LIN {X -286.815,Y -42.863,Z 84.157,A 8.500,B 90.000,C 0.000} C_DIS
LIN {X -286.571,Y -44.464,Z 82.253,A 8.820,B 90.000,C 0.000} C_DIS
LIN {X -286.317,Y -46.071,Z 80.355,A 9.141,B 90.000,C 0.000} C_DIS
LIN {X -286.054,Y -47.677,Z 78.457,A 9.463,B 90.000,C 0.000} C_DIS
LIN {X -285.784,Y -49.269,Z 76.549,A 9.782,B 90.000,C 0.000} C_DIS
LIN {X -285.503,Y -50.872,Z 74.651,A 10.103,B 90.000,C 0.000} C_DIS
LIN {X -285.213,Y -52.473,Z 72.753,A 10.425,B 90.000,C 0.000} C_DIS
LIN {X -284.916,Y -54.061,Z 70.845,A 10.744,B 90.000,C 0.000} C_DIS
LIN {X -284.609,Y -55.658,Z 68.946,A 11.065,B 90.000,C 0.000} C_DIS
LIN {X -284.292,Y -57.253,Z 67.048,A 11.386,B 90.000,C 0.000} C_DIS
LIN {X -284.017,Y -58.605,Z 65.403,A 11.659,B 90.000,C 0.000} C_DIS
LIN {X -283.964,Y -58.859,Z 65.202,A 11.710,B 90.000,C 0.000} C_DIS
LIN {X -283.906,Y -59.138,Z 65.153,A 11.767,B 90.000,C 0.000} C_DIS
LIN {X -283.848,Y -59.418,Z 65.202,A 11.823,B 90.000,C 0.000} C_DIS
LIN {X -283.795,Y -59.671,Z 65.403,A 11.874,B 90.000,C 0.000} C_DIS
LIN {X -283.751,Y -59.880,Z 65.687,A 11.916,B 90.000,C 0.000} C_DIS
LIN {X -283.739,Y -59.937,Z 66.462,A 11.928,B 90.000,C 0.000} C_DIS
LIN {X -283.717,Y -60.038,Z 66.779,A 11.948,B 90.000,C 0.000} C_DIS
LIN {X -283.709,Y -60.077,Z 67.718,A 11.956,B 90.000,C 0.000} C_DIS
LIN {X -283.687,Y -60.180,Z 68.098,A 11.977,B 90.000,C 0.000} C_DIS
LIN {X -283.679,Y -60.218,Z 69.146,A 11.985,B 90.000,C 0.000} C_DIS
LIN {X -283.657,Y -60.321,Z 69.525,A 12.005,B 90.000,C 0.000} C_DIS
LIN {X -283.649,Y -60.360,Z 70.464,A 12.013,B 90.000,C 0.000} C_DIS
LIN {X -283.627,Y -60.462,Z 70.826,A 12.034,B 90.000,C 0.000} C_DIS
LIN {X -283.619,Y -60.501,Z 71.765,A 12.042,B 90.000,C 0.000} C_DIS
LIN {X -283.597,Y -60.603,Z 72.126,A 12.062,B 90.000,C 0.000} C_DIS
LIN {X -283.589,Y -60.643,Z 73.066,A 12.070,B 90.000,C 0.000} C_DIS
LIN {X -283.567,Y -60.745,Z 73.445,A 12.091,B 90.000,C 0.000} C_DIS
LIN {X -283.558,Y -60.784,Z 74.493,A 12.099,B 90.000,C 0.000} C_DIS
LIN {X -283.536,Y -60.886,Z 74.872,A 12.120,B 90.000,C 0.000} C_DIS
LIN {X -283.528,Y -60.925,Z 75.812,A 12.127,B 90.000,C 0.000} C_DIS
LIN {X -283.506,Y -61.028,Z 76.191,A 12.148,B 90.000,C 0.000} C_DIS
LIN {X -283.498,Y -61.066,Z 77.239,A 12.156,B 90.000,C 0.000} C_DIS
LIN {X -283.476,Y -61.169,Z 77.618,A 12.177,B 90.000,C 0.000} C_DIS
LIN {X -283.467,Y -61.208,Z 78.558,A 12.185,B 90.000,C 0.000} C_DIS
LIN {X -283.445,Y -61.310,Z 78.919,A 12.205,B 90.000,C 0.000} C_DIS
LIN {X -283.437,Y -61.349,Z 79.859,A 12.213,B 90.000,C 0.000} C_DIS
LIN {X -283.414,Y -61.451,Z 80.220,A 12.234,B 90.000,C 0.000} C_DIS
LIN {X -283.406,Y -61.490,Z 81.159,A 12.242,B 90.000,C 0.000} C_DIS
LIN {X -283.384,Y -61.592,Z 81.521,A 12.262,B 90.000,C 0.000} C_DIS
LIN {X -283.375,Y -61.632,Z 82.460,A 12.270,B 90.000,C 0.000} C_DIS
LIN {X -283.353,Y -61.734,Z 82.840,A 12.291,B 90.000,C 0.000} C_DIS
LIN {X -283.345,Y -61.773,Z 83.887,A 12.299,B 90.000,C 0.000} C_DIS
LIN {X -283.322,Y -61.875,Z 84.267,A 12.319,B 90.000,C 0.000} C_DIS
LIN {X -283.314,Y -61.914,Z 85.206,A 12.327,B 90.000,C 0.000} C_DIS
LIN {X -283.291,Y -62.016,Z 85.586,A 12.348,B 90.000,C 0.000} C_DIS
LIN {X -283.283,Y -62.055,Z 86.633,A 12.356,B 90.000,C 0.000} C_DIS
LIN {X -283.260,Y -62.157,Z 87.013,A 12.377,B 90.000,C 0.000} C_DIS
LIN {X -283.252,Y -62.196,Z 87.952,A 12.384,B 90.000,C 0.000} C_DIS
LIN {X -283.229,Y -62.298,Z 88.314,A 12.405,B 90.000,C 0.000} C_DIS
LIN {X -283.221,Y -62.338,Z 89.253,A 12.413,B 90.000,C 0.000} C_DIS
LIN {X -283.198,Y -62.440,Z 89.614,A 12.434,B 90.000,C 0.000} C_DIS
LIN {X -283.190,Y -62.479,Z 90.554,A 12.442,B 90.000,C 0.000} C_DIS
LIN {X -283.167,Y -62.581,Z 90.933,A 12.462,B 90.000,C 0.000} C_DIS
LIN {X -283.159,Y -62.620,Z 91.981,A 12.470,B 90.000,C 0.000} C_DIS
LIN {X -283.136,Y -62.722,Z 92.360,A 12.491,B 90.000,C 0.000} C_DIS
LIN {X -283.127,Y -62.761,Z 93.300,A 12.499,B 90.000,C 0.000} C_DIS
LIN {X -283.105,Y -62.863,Z 93.661,A 12.519,B 90.000,C 0.000} C_DIS
LIN {X -283.096,Y -62.902,Z 94.601,A 12.527,B 90.000,C 0.000} C_DIS
LIN {X -283.073,Y -63.004,Z 94.962,A 12.548,B 90.000,C 0.000} C_DIS
LIN {X -283.065,Y -63.043,Z 95.901,A 12.556,B 90.000,C 0.000} C_DIS
LIN {X -283.042,Y -63.145,Z 96.281,A 12.576,B 90.000,C 0.000} C_DIS
LIN {X -283.033,Y -63.184,Z 97.329,A 12.584,B 90.000,C 0.000} C_DIS
LIN {X -283.010,Y -63.286,Z 97.708,A 12.605,B 90.000,C 0.000} C_DIS
LIN {X -283.002,Y -63.325,Z 98.647,A 12.613,B 90.000,C 0.000} C_DIS
LIN {X -282.979,Y -63.427,Z 99.009,A 12.634,B 90.000,C 0.000} C_DIS
LIN {X -282.970,Y -63.466,Z 99.948,A 12.641,B 90.000,C 0.000} C_DIS
LIN {X -282.947,Y -63.568,Z 100.309,A 12.662,B 90.000,C 0.000} C_DIS
LIN {X -282.938,Y -63.607,Z 101.249,A 12.670,B 90.000,C 0.000} C_DIS
LIN {X -282.915,Y -63.709,Z 101.628,A 12.691,B 90.000,C 0.000} C_DIS
LIN {X -282.907,Y -63.748,Z 102.676,A 12.699,B 90.000,C 0.000} C_DIS
LIN {X -282.884,Y -63.850,Z 103.055,A 12.719,B 90.000,C 0.000} C_DIS
LIN {X -282.875,Y -63.889,Z 103.995,A 12.727,B 90.000,C 0.000} C_DIS
LIN {X -282.852,Y -63.991,Z 104.356,A 12.748,B 90.000,C 0.000} C_DIS
LIN {X -282.843,Y -64.030,Z 105.296,A 12.756,B 90.000,C 0.000} C_DIS
LIN {X -282.820,Y -64.132,Z 105.657,A 12.776,B 90.000,C 0.000} C_DIS
LIN {X -282.811,Y -64.171,Z 106.596,A 12.784,B 90.000,C 0.000} C_DIS
LIN {X -282.788,Y -64.273,Z 106.976,A 12.805,B 90.000,C 0.000} C_DIS
LIN {X -282.779,Y -64.312,Z 108.024,A 12.813,B 90.000,C 0.000} C_DIS
LIN {X -282.756,Y -64.414,Z 108.403,A 12.833,B 90.000,C 0.000} C_DIS
LIN {X -282.747,Y -64.453,Z 109.342,A 12.841,B 90.000,C 0.000} C_DIS
LIN {X -282.724,Y -64.555,Z 109.722,A 12.862,B 90.000,C 0.000} C_DIS
LIN {X -282.715,Y -64.594,Z 110.770,A 12.870,B 90.000,C 0.000} C_DIS
LIN {X -282.691,Y -64.696,Z 111.149,A 12.891,B 90.000,C 0.000} C_DIS
LIN {X -282.682,Y -64.735,Z 112.089,A 12.898,B 90.000,C 0.000} C_DIS
LIN {X -282.659,Y -64.837,Z 112.450,A 12.919,B 90.000,C 0.000} C_DIS
LIN {X -282.650,Y -64.876,Z 113.389,A 12.927,B 90.000,C 0.000} C_DIS
LIN {X -282.627,Y -64.978,Z 113.751,A 12.948,B 90.000,C 0.000} C_DIS
LIN {X -282.618,Y -65.017,Z 114.690,A 12.956,B 90.000,C 0.000} C_DIS
LIN {X -282.594,Y -65.118,Z 115.051,A 12.976,B 90.000,C 0.000} C_DIS
LIN {X -282.585,Y -65.157,Z 115.991,A 12.984,B 90.000,C 0.000} C_DIS
LIN {X -282.562,Y -65.259,Z 116.370,A 13.005,B 90.000,C 0.000} C_DIS
LIN {X -282.553,Y -65.298,Z 117.418,A 13.013,B 90.000,C 0.000} C_DIS
LIN {X -282.529,Y -65.400,Z 117.797,A 13.033,B 90.000,C 0.000} C_DIS
LIN {X -282.520,Y -65.439,Z 118.737,A 13.041,B 90.000,C 0.000} C_DIS
LIN {X -282.497,Y -65.541,Z 119.098,A 13.062,B 90.000,C 0.000} C_DIS
LIN {X -282.488,Y -65.580,Z 120.038,A 13.070,B 90.000,C 0.000} C_DIS
LIN {X -282.464,Y -65.682,Z 120.417,A 13.090,B 90.000,C 0.000} C_DIS
LIN {X -282.455,Y -65.720,Z 121.465,A 13.098,B 90.000,C 0.000} C_DIS
LIN {X -282.431,Y -65.822,Z 121.844,A 13.119,B 90.000,C 0.000} C_DIS
LIN {X -282.422,Y -65.861,Z 122.784,A 13.127,B 90.000,C 0.000} C_DIS
LIN {X -282.398,Y -65.963,Z 123.145,A 13.148,B 90.000,C 0.000} C_DIS
LIN {X -282.389,Y -66.002,Z 124.084,A 13.155,B 90.000,C 0.000} C_DIS
LIN {X -282.365,Y -66.104,Z 124.464,A 13.176,B 90.000,C 0.000} C_DIS
LIN {X -282.356,Y -66.143,Z 125.512,A 13.184,B 90.000,C 0.000} C_DIS
LIN {X -282.333,Y -66.245,Z 125.891,A 13.205,B 90.000,C 0.000} C_DIS
LIN {X -282.323,Y -66.284,Z 126.830,A 13.213,B 90.000,C 0.000} C_DIS
LIN {X -282.299,Y -66.385,Z 127.192,A 13.233,B 90.000,C 0.000} C_DIS
LIN {X -282.290,Y -66.424,Z 128.131,A 13.241,B 90.000,C 0.000} C_DIS
LIN {X -282.266,Y -66.526,Z 128.492,A 13.262,B 90.000,C 0.000} C_DIS
LIN {X -282.257,Y -66.565,Z 129.432,A 13.270,B 90.000,C 0.000} C_DIS
LIN {X -282.233,Y -66.667,Z 129.811,A 13.290,B 90.000,C 0.000} C_DIS
LIN {X -282.224,Y -66.705,Z 130.859,A 13.298,B 90.000,C 0.000} C_DIS
LIN {X -282.200,Y -66.807,Z 131.239,A 13.319,B 90.000,C 0.000} C_DIS
LIN {X -282.191,Y -66.846,Z 132.178,A 13.327,B 90.000,C 0.000} C_DIS
LIN {X -282.167,Y -66.948,Z 132.539,A 13.347,B 90.000,C 0.000} C_DIS
LIN {X -282.157,Y -66.987,Z 133.479,A 13.355,B 90.000,C 0.000} C_DIS
LIN {X -282.133,Y -67.089,Z 133.858,A 13.376,B 90.000,C 0.000} C_DIS
LIN {X -282.124,Y -67.127,Z 134.906,A 13.384,B 90.000,C 0.000} C_DIS
LIN {X -282.100,Y -67.229,Z 135.285,A 13.405,B 90.000,C 0.000} C_DIS
LIN {X -282.090,Y -67.268,Z 136.225,A 13.412,B 90.000,C 0.000} C_DIS
LIN {X -282.066,Y -67.370,Z 136.586,A 13.433,B 90.000,C 0.000} C_DIS
LIN {X -282.057,Y -67.409,Z 137.525,A 13.441,B 90.000,C 0.000} C_DIS
LIN {X -282.033,Y -67.510,Z 137.887,A 13.462,B 90.000,C 0.000} C_DIS
LIN {X -282.023,Y -67.549,Z 138.826,A 13.470,B 90.000,C 0.000} C_DIS
LIN {X -281.999,Y -67.651,Z 139.206,A 13.490,B 90.000,C 0.000} C_DIS
LIN {X -281.990,Y -67.690,Z 140.253,A 13.498,B 90.000,C 0.000} C_DIS
LIN {X -281.965,Y -67.791,Z 140.633,A 13.519,B 90.000,C 0.000} C_DIS
LIN {X -281.956,Y -67.830,Z 141.572,A 13.527,B 90.000,C 0.000} C_DIS
LIN {X -281.931,Y -67.932,Z 141.934,A 13.547,B 90.000,C 0.000} C_DIS
LIN {X -281.922,Y -67.971,Z 142.873,A 13.555,B 90.000,C 0.000} C_DIS
LIN {X -281.897,Y -68.073,Z 143.252,A 13.576,B 90.000,C 0.000} C_DIS
LIN {X -281.888,Y -68.111,Z 144.300,A 13.584,B 90.000,C 0.000} C_DIS
LIN {X -281.863,Y -68.213,Z 144.680,A 13.604,B 90.000,C 0.000} C_DIS
LIN {X -281.854,Y -68.252,Z 145.619,A 13.612,B 90.000,C 0.000} C_DIS
LIN {X -281.829,Y -68.353,Z 145.980,A 13.633,B 90.000,C 0.000} C_DIS
LIN {X -281.820,Y -68.392,Z 146.920,A 13.641,B 90.000,C 0.000} C_DIS
LIN {X -281.795,Y -68.494,Z 147.281,A 13.662,B 90.000,C 0.000} C_DIS
LIN {X -281.786,Y -68.533,Z 148.221,A 13.669,B 90.000,C 0.000} C_DIS
LIN {X -281.761,Y -68.635,Z 148.618,A 13.690,B 90.000,C 0.000} C_DIS
LIN {X -281.761,Y -68.635,Z 149.774,A 13.690,B 90.000,C 0.000} C_DIS
LIN {X -281.774,Y -68.583,Z 149.991,A 13.680,B 90.000,C 0.000} C_DIS
LIN {X -281.786,Y -68.533,Z 150.136,A 13.670,B 90.000,C 0.000} C_DIS
LIN {X -281.795,Y -68.493,Z 150.858,A 13.661,B 90.000,C 0.000} C_DIS
LIN {X -281.820,Y -68.393,Z 151.147,A 13.641,B 90.000,C 0.000} C_DIS
LIN {X -281.830,Y -68.353,Z 151.870,A 13.633,B 90.000,C 0.000} C_DIS
LIN {X -281.854,Y -68.252,Z 152.159,A 13.612,B 90.000,C 0.000} C_DIS
LIN {X -281.864,Y -68.212,Z 152.882,A 13.604,B 90.000,C 0.000} C_DIS
LIN {X -281.888,Y -68.112,Z 153.171,A 13.584,B 90.000,C 0.000} C_DIS
LIN {X -281.898,Y -68.072,Z 153.893,A 13.576,B 90.000,C 0.000} C_DIS
LIN {X -281.922,Y -67.971,Z 154.182,A 13.555,B 90.000,C 0.000} C_DIS
LIN {X -281.931,Y -67.931,Z 154.905,A 13.547,B 90.000,C 0.000} C_DIS
LIN {X -281.956,Y -67.831,Z 155.194,A 13.527,B 90.000,C 0.000} C_DIS
LIN {X -281.965,Y -67.791,Z 155.917,A 13.519,B 90.000,C 0.000} C_DIS
LIN {X -281.989,Y -67.690,Z 156.206,A 13.498,B 90.000,C 0.000} C_DIS
LIN {X -281.999,Y -67.650,Z 156.928,A 13.490,B 90.000,C 0.000} C_DIS
LIN {X -282.023,Y -67.550,Z 157.217,A 13.470,B 90.000,C 0.000} C_DIS
LIN {X -282.033,Y -67.510,Z 157.940,A 13.462,B 90.000,C 0.000} C_DIS
LIN {X -282.057,Y -67.409,Z 158.229,A 13.441,B 90.000,C 0.000} C_DIS
LIN {X -282.066,Y -67.369,Z 158.952,A 13.433,B 90.000,C 0.000} C_DIS
LIN {X -282.090,Y -67.269,Z 159.241,A 13.413,B 90.000,C 0.000} C_DIS
LIN {X -282.100,Y -67.229,Z 159.963,A 13.404,B 90.000,C 0.000} C_DIS
LIN {X -282.124,Y -67.128,Z 160.253,A 13.384,B 90.000,C 0.000} C_DIS
LIN {X -282.133,Y -67.088,Z 160.975,A 13.376,B 90.000,C 0.000} C_DIS
LIN {X -282.157,Y -66.987,Z 161.264,A 13.355,B 90.000,C 0.000} C_DIS
LIN {X -282.167,Y -66.947,Z 161.987,A 13.347,B 90.000,C 0.000} C_DIS
LIN {X -282.191,Y -66.847,Z 162.276,A 13.327,B 90.000,C 0.000} C_DIS
LIN {X -282.200,Y -66.807,Z 162.999,A 13.319,B 90.000,C 0.000} C_DIS
LIN {X -282.224,Y -66.706,Z 163.288,A 13.298,B 90.000,C 0.000} C_DIS
LIN {X -282.233,Y -66.666,Z 164.010,A 13.290,B 90.000,C 0.000} C_DIS
LIN {X -282.257,Y -66.566,Z 164.299,A 13.270,B 90.000,C 0.000} C_DIS
LIN {X -282.266,Y -66.525,Z 165.022,A 13.262,B 90.000,C 0.000} C_DIS
LIN {X -282.290,Y -66.425,Z 165.311,A 13.241,B 90.000,C 0.000} C_DIS
LIN {X -282.300,Y -66.385,Z 166.034,A 13.233,B 90.000,C 0.000} C_DIS
LIN {X -282.323,Y -66.285,Z 166.305,A 13.213,B 90.000,C 0.000} C_DIS
LIN {X -282.333,Y -66.244,Z 166.919,A 13.204,B 90.000,C 0.000} C_DIS
LIN {X -282.356,Y -66.143,Z 167.190,A 13.184,B 90.000,C 0.000} C_DIS
LIN {X -282.366,Y -66.103,Z 167.913,A 13.176,B 90.000,C 0.000} C_DIS
LIN {X -282.389,Y -66.002,Z 168.220,A 13.155,B 90.000,C 0.000} C_DIS
LIN {X -282.398,Y -65.963,Z 169.051,A 13.147,B 90.000,C 0.000} C_DIS
LIN {X -282.422,Y -65.862,Z 169.358,A 13.127,B 90.000,C 0.000} C_DIS
LIN {X -282.431,Y -65.822,Z 170.080,A 13.119,B 90.000,C 0.000} C_DIS
LIN {X -282.455,Y -65.721,Z 170.370,A 13.098,B 90.000,C 0.000} C_DIS
LIN {X -282.464,Y -65.681,Z 171.092,A 13.090,B 90.000,C 0.000} C_DIS
LIN {X -282.488,Y -65.580,Z 171.381,A 13.070,B 90.000,C 0.000} C_DIS
LIN {X -282.497,Y -65.540,Z 172.104,A 13.062,B 90.000,C 0.000} C_DIS
LIN {X -282.520,Y -65.440,Z 172.375,A 13.041,B 90.000,C 0.000} C_DIS
LIN {X -282.530,Y -65.399,Z 172.989,A 13.033,B 90.000,C 0.000} C_DIS
LIN {X -282.553,Y -65.299,Z 173.260,A 13.013,B 90.000,C 0.000} C_DIS
LIN {X -282.562,Y -65.259,Z 173.983,A 13.005,B 90.000,C 0.000} C_DIS
LIN {X -282.585,Y -65.158,Z 174.272,A 12.984,B 90.000,C 0.000} C_DIS
LIN {X -282.595,Y -65.118,Z 174.994,A 12.976,B 90.000,C 0.000} C_DIS
LIN {X -282.618,Y -65.017,Z 175.283,A 12.956,B 90.000,C 0.000} C_DIS
LIN {X -282.627,Y -64.977,Z 176.006,A 12.948,B 90.000,C 0.000} C_DIS
LIN {X -282.650,Y -64.876,Z 176.295,A 12.927,B 90.000,C 0.000} C_DIS
LIN {X -282.659,Y -64.836,Z 177.018,A 12.919,B 90.000,C 0.000} C_DIS
LIN {X -282.682,Y -64.735,Z 177.307,A 12.899,B 90.000,C 0.000} C_DIS
LIN {X -282.692,Y -64.695,Z 178.030,A 12.890,B 90.000,C 0.000} C_DIS
LIN {X -282.715,Y -64.595,Z 178.319,A 12.870,B 90.000,C 0.000} C_DIS
LIN {X -282.724,Y -64.554,Z 179.041,A 12.862,B 90.000,C 0.000} C_DIS
LIN {X -282.747,Y -64.454,Z 179.330,A 12.841,B 90.000,C 0.000} C_DIS
LIN {X -282.756,Y -64.413,Z 180.053,A 12.833,B 90.000,C 0.000} C_DIS
LIN {X -282.779,Y -64.313,Z 180.342,A 12.813,B 90.000,C 0.000} C_DIS
LIN {X -282.788,Y -64.272,Z 181.065,A 12.805,B 90.000,C 0.000} C_DIS
LIN {X -282.811,Y -64.172,Z 181.354,A 12.784,B 90.000,C 0.000} C_DIS
LIN {X -282.820,Y -64.132,Z 182.076,A 12.776,B 90.000,C 0.000} C_DIS
LIN {X -282.843,Y -64.031,Z 182.365,A 12.756,B 90.000,C 0.000} C_DIS
LIN {X -282.852,Y -63.991,Z 183.088,A 12.748,B 90.000,C 0.000} C_DIS
LIN {X -282.875,Y -63.890,Z 183.377,A 12.727,B 90.000,C 0.000} C_DIS
LIN {X -282.884,Y -63.850,Z 184.100,A 12.719,B 90.000,C 0.000} C_DIS
LIN {X -282.906,Y -63.749,Z 184.389,A 12.699,B 90.000,C 0.000} C_DIS
LIN {X -282.916,Y -63.709,Z 185.111,A 12.691,B 90.000,C 0.000} C_DIS
LIN {X -282.938,Y -63.608,Z 185.400,A 12.670,B 90.000,C 0.000} C_DIS
LIN {X -282.947,Y -63.568,Z 186.123,A 12.662,B 90.000,C 0.000} C_DIS
LIN {X -282.970,Y -63.467,Z 186.412,A 12.642,B 90.000,C 0.000} C_DIS
LIN {X -282.979,Y -63.427,Z 187.135,A 12.633,B 90.000,C 0.000} C_DIS
LIN {X -283.001,Y -63.326,Z 187.424,A 12.613,B 90.000,C 0.000} C_DIS
LIN {X -283.010,Y -63.286,Z 188.146,A 12.605,B 90.000,C 0.000} C_DIS
LIN {X -283.033,Y -63.185,Z 188.436,A 12.584,B 90.000,C 0.000} C_DIS
LIN {X -283.042,Y -63.145,Z 189.158,A 12.576,B 90.000,C 0.000} C_DIS
LIN {X -283.064,Y -63.044,Z 189.447,A 12.556,B 90.000,C 0.000} C_DIS
LIN {X -283.073,Y -63.003,Z 190.170,A 12.548,B 90.000,C 0.000} C_DIS
LIN {X -283.096,Y -62.903,Z 190.459,A 12.527,B 90.000,C 0.000} C_DIS
LIN {X -283.105,Y -62.862,Z 191.182,A 12.519,B 90.000,C 0.000} C_DIS
LIN {X -283.127,Y -62.762,Z 191.471,A 12.499,B 90.000,C 0.000} C_DIS
LIN {X -283.136,Y -62.721,Z 192.193,A 12.491,B 90.000,C 0.000} C_DIS
LIN {X -283.158,Y -62.620,Z 192.482,A 12.470,B 90.000,C 0.000} C_DIS
LIN {X -283.167,Y -62.580,Z 193.205,A 12.462,B 90.000,C 0.000} C_DIS
LIN {X -283.190,Y -62.479,Z 193.494,A 12.442,B 90.000,C 0.000} C_DIS
LIN {X -283.198,Y -62.439,Z 194.217,A 12.434,B 90.000,C 0.000} C_DIS
LIN {X -283.221,Y -62.338,Z 194.506,A 12.413,B 90.000,C 0.000} C_DIS
LIN {X -283.230,Y -62.298,Z 195.228,A 12.405,B 90.000,C 0.000} C_DIS
LIN {X -283.252,Y -62.197,Z 195.517,A 12.385,B 90.000,C 0.000} C_DIS
LIN {X -283.261,Y -62.157,Z 196.240,A 12.376,B 90.000,C 0.000} C_DIS
LIN {X -283.283,Y -62.056,Z 196.529,A 12.356,B 90.000,C 0.000} C_DIS
LIN {X -283.291,Y -62.016,Z 197.252,A 12.348,B 90.000,C 0.000} C_DIS
LIN {X -283.314,Y -61.915,Z 197.541,A 12.327,B 90.000,C 0.000} C_DIS
LIN {X -283.322,Y -61.874,Z 198.263,A 12.319,B 90.000,C 0.000} C_DIS
LIN {X -283.344,Y -61.773,Z 198.553,A 12.299,B 90.000,C 0.000} C_DIS
LIN {X -283.353,Y -61.733,Z 199.275,A 12.291,B 90.000,C 0.000} C_DIS
LIN {X -283.375,Y -61.632,Z 199.564,A 12.270,B 90.000,C 0.000} C_DIS
LIN {X -283.384,Y -61.592,Z 200.287,A 12.262,B 90.000,C 0.000} C_DIS
LIN {X -283.406,Y -61.491,Z 200.576,A 12.242,B 90.000,C 0.000} C_DIS
LIN {X -283.415,Y -61.451,Z 201.299,A 12.234,B 90.000,C 0.000} C_DIS
LIN {X -283.436,Y -61.350,Z 201.588,A 12.213,B 90.000,C 0.000} C_DIS
LIN {X -283.445,Y -61.309,Z 202.310,A 12.205,B 90.000,C 0.000} C_DIS
LIN {X -283.467,Y -61.209,Z 202.599,A 12.185,B 90.000,C 0.000} C_DIS
LIN {X -283.476,Y -61.168,Z 203.322,A 12.177,B 90.000,C 0.000} C_DIS
LIN {X -283.497,Y -61.067,Z 203.611,A 12.156,B 90.000,C 0.000} C_DIS
LIN {X -283.506,Y -61.027,Z 204.334,A 12.148,B 90.000,C 0.000} C_DIS
LIN {X -283.528,Y -60.926,Z 204.623,A 12.128,B 90.000,C 0.000} C_DIS
LIN {X -283.537,Y -60.886,Z 205.345,A 12.119,B 90.000,C 0.000} C_DIS
LIN {X -283.558,Y -60.785,Z 205.634,A 12.099,B 90.000,C 0.000} C_DIS
LIN {X -283.567,Y -60.744,Z 206.357,A 12.091,B 90.000,C 0.000} C_DIS
LIN {X -283.588,Y -60.643,Z 206.646,A 12.070,B 90.000,C 0.000} C_DIS
LIN {X -283.597,Y -60.603,Z 207.369,A 12.062,B 90.000,C 0.000} C_DIS
LIN {X -283.619,Y -60.502,Z 207.658,A 12.042,B 90.000,C 0.000} C_DIS
LIN {X -283.627,Y -60.462,Z 208.380,A 12.034,B 90.000,C 0.000} C_DIS
LIN {X -283.649,Y -60.361,Z 208.670,A 12.013,B 90.000,C 0.000} C_DIS
LIN {X -283.657,Y -60.320,Z 209.392,A 12.005,B 90.000,C 0.000} C_DIS
LIN {X -283.679,Y -60.219,Z 209.681,A 11.985,B 90.000,C 0.000} C_DIS
LIN {X -283.687,Y -60.179,Z 210.404,A 11.977,B 90.000,C 0.000} C_DIS
LIN {X -283.709,Y -60.078,Z 210.693,A 11.956,B 90.000,C 0.000} C_DIS
LIN {X -283.717,Y -60.037,Z 211.416,A 11.948,B 90.000,C 0.000} C_DIS
LIN {X -283.739,Y -59.937,Z 211.687,A 11.928,B 90.000,C 0.000} C_DIS
LIN {X -283.747,Y -59.896,Z 212.301,A 11.919,B 90.000,C 0.000} C_DIS
LIN {X -283.769,Y -59.795,Z 212.590,A 11.899,B 90.000,C 0.000} C_DIS
LIN {X -283.777,Y -59.755,Z 213.421,A 11.891,B 90.000,C 0.000} C_DIS
LIN {X -283.798,Y -59.654,Z 213.710,A 11.871,B 90.000,C 0.000} C_DIS
LIN {X -283.807,Y -59.613,Z 214.324,A 11.862,B 90.000,C 0.000} C_DIS
LIN {X -283.828,Y -59.512,Z 214.613,A 11.842,B 90.000,C 0.000} C_DIS
LIN {X -283.836,Y -59.472,Z 215.444,A 11.834,B 90.000,C 0.000} C_DIS
LIN {X -283.858,Y -59.371,Z 215.751,A 11.813,B 90.000,C 0.000} C_DIS
LIN {X -283.866,Y -59.330,Z 216.474,A 11.805,B 90.000,C 0.000} C_DIS
LIN {X -283.887,Y -59.229,Z 216.763,A 11.785,B 90.000,C 0.000} C_DIS
LIN {X -283.896,Y -59.189,Z 217.486,A 11.777,B 90.000,C 0.000} C_DIS
LIN {X -283.917,Y -59.088,Z 217.775,A 11.756,B 90.000,C 0.000} C_DIS
LIN {X -283.925,Y -59.047,Z 218.497,A 11.748,B 90.000,C 0.000} C_DIS
LIN {X -283.946,Y -58.946,Z 218.786,A 11.728,B 90.000,C 0.000} C_DIS
LIN {X -283.954,Y -58.906,Z 219.509,A 11.720,B 90.000,C 0.000} C_DIS
LIN {X -283.975,Y -58.805,Z 219.780,A 11.699,B 90.000,C 0.000} C_DIS
LIN {X -283.984,Y -58.764,Z 220.394,A 11.691,B 90.000,C 0.000} C_DIS
LIN {X -284.005,Y -58.663,Z 220.665,A 11.671,B 90.000,C 0.000} C_DIS
LIN {X -284.013,Y -58.623,Z 221.388,A 11.663,B 90.000,C 0.000} C_DIS
LIN {X -284.034,Y -58.522,Z 221.677,A 11.642,B 90.000,C 0.000} C_DIS
LIN {X -284.042,Y -58.481,Z 222.400,A 11.634,B 90.000,C 0.000} C_DIS
LIN {X -284.063,Y -58.380,Z 222.689,A 11.614,B 90.000,C 0.000} C_DIS
LIN {X -284.071,Y -58.340,Z 223.411,A 11.605,B 90.000,C 0.000} C_DIS
LIN {X -284.092,Y -58.239,Z 223.700,A 11.585,B 90.000,C 0.000} C_DIS
LIN {X -284.100,Y -58.198,Z 224.423,A 11.577,B 90.000,C 0.000} C_DIS
LIN {X -284.121,Y -58.097,Z 224.712,A 11.557,B 90.000,C 0.000} C_DIS
LIN {X -284.129,Y -58.056,Z 225.435,A 11.548,B 90.000,C 0.000} C_DIS
LIN {X -284.150,Y -57.955,Z 225.724,A 11.528,B 90.000,C 0.000} C_DIS
LIN {X -284.158,Y -57.915,Z 226.446,A 11.520,B 90.000,C 0.000} C_DIS
LIN {X -284.179,Y -57.814,Z 226.736,A 11.499,B 90.000,C 0.000} C_DIS
LIN {X -284.187,Y -57.773,Z 227.458,A 11.491,B 90.000,C 0.000} C_DIS
LIN {X -284.208,Y -57.672,Z 227.747,A 11.471,B 90.000,C 0.000} C_DIS
LIN {X -284.216,Y -57.632,Z 228.470,A 11.463,B 90.000,C 0.000} C_DIS
LIN {X -284.236,Y -57.530,Z 228.759,A 11.442,B 90.000,C 0.000} C_DIS
LIN {X -284.244,Y -57.490,Z 229.482,A 11.434,B 90.000,C 0.000} C_DIS
LIN {X -284.265,Y -57.389,Z 229.771,A 11.414,B 90.000,C 0.000} C_DIS
LIN {X -284.273,Y -57.348,Z 230.493,A 11.406,B 90.000,C 0.000} C_DIS
LIN {X -284.293,Y -57.247,Z 230.782,A 11.385,B 90.000,C 0.000} C_DIS
LIN {X -284.302,Y -57.207,Z 231.505,A 11.377,B 90.000,C 0.000} C_DIS
LIN {X -284.322,Y -57.105,Z 231.794,A 11.357,B 90.000,C 0.000} C_DIS
LIN {X -284.330,Y -57.065,Z 232.517,A 11.348,B 90.000,C 0.000} C_DIS
LIN {X -284.350,Y -56.964,Z 232.806,A 11.328,B 90.000,C 0.000} C_DIS
LIN {X -284.358,Y -56.923,Z 233.528,A 11.320,B 90.000,C 0.000} C_DIS
LIN {X -284.379,Y -56.822,Z 233.817,A 11.300,B 90.000,C 0.000} C_DIS
LIN {X -284.387,Y -56.781,Z 234.540,A 11.291,B 90.000,C 0.000} C_DIS
LIN {X -284.407,Y -56.680,Z 234.829,A 11.271,B 90.000,C 0.000} C_DIS
LIN {X -284.415,Y -56.640,Z 235.552,A 11.263,B 90.000,C 0.000} C_DIS
LIN {X -284.425,Y -56.589,Z 235.696,A 11.253,B 90.000,C 0.000} C_DIS
LIN {X -284.435,Y -56.539,Z 235.772,A 11.243,B 90.000,C 0.000} C_DIS
LIN {X -284.448,Y -56.472,Z 236.202,A 11.229,B 90.000,C 0.000} C_DIS
LIN {X -284.474,Y -56.342,Z 236.395,A 11.203,B 90.000,C 0.000} C_DIS
LIN {X -284.514,Y -56.141,Z 236.519,A 11.162,B 90.000,C 0.000} C_DIS
LIN {X -284.565,Y -55.882,Z 236.563,A 11.110,B 90.000,C 0.000} C_DIS
LIN {X -284.623,Y -55.588,Z 236.506,A 11.051,B 90.000,C 0.000} C_DIS
LIN {X -284.683,Y -55.275,Z 236.240,A 10.988,B 90.000,C 0.000} C_DIS
LIN {X -284.727,Y -55.051,Z 235.979,A 10.943,B 90.000,C 0.000} C_DIS
LIN {X -284.745,Y -54.958,Z 235.807,A 10.924,B 90.000,C 0.000} C_DIS
LIN {X -284.749,Y -54.937,Z 235.729,A 10.920,B 90.000,C 0.000} C_DIS
LIN {X -284.768,Y -54.837,Z 235.659,A 10.900,B 90.000,C 0.000} C_DIS
LIN {X -284.772,Y -54.816,Z 235.568,A 10.896,B 90.000,C 0.000} C_DIS
LIN {X -284.780,Y -54.774,Z 235.446,A 10.887,B 90.000,C 0.000} C_DIS
LIN {X -284.819,Y -54.574,Z 235.228,A 10.847,B 90.000,C 0.000} C_DIS
LIN {X -284.835,Y -54.491,Z 235.008,A 10.830,B 90.000,C 0.000} C_DIS
LIN {X -284.873,Y -54.290,Z 234.795,A 10.790,B 90.000,C 0.000} C_DIS
LIN {X -284.889,Y -54.207,Z 234.574,A 10.773,B 90.000,C 0.000} C_DIS
LIN {X -284.927,Y -54.006,Z 234.361,A 10.733,B 90.000,C 0.000} C_DIS
LIN {X -284.943,Y -53.923,Z 234.141,A 10.716,B 90.000,C 0.000} C_DIS
LIN {X -284.981,Y -53.722,Z 233.928,A 10.676,B 90.000,C 0.000} C_DIS
LIN {X -284.996,Y -53.639,Z 233.707,A 10.659,B 90.000,C 0.000} C_DIS
LIN {X -285.034,Y -53.438,Z 233.489,A 10.619,B 90.000,C 0.000} C_DIS
LIN {X -285.042,Y -53.396,Z 233.368,A 10.610,B 90.000,C 0.000} C_DIS
LIN {X -285.046,Y -53.375,Z 233.277,A 10.606,B 90.000,C 0.000} C_DIS
LIN {X -285.065,Y -53.275,Z 233.202,A 10.586,B 90.000,C 0.000} C_DIS
LIN {X -285.068,Y -53.254,Z 233.111,A 10.582,B 90.000,C 0.000} C_DIS
LIN {X -285.076,Y -53.212,Z 232.989,A 10.573,B 90.000,C 0.000} C_DIS
LIN {X -285.114,Y -53.012,Z 232.771,A 10.533,B 90.000,C 0.000} C_DIS
LIN {X -285.129,Y -52.928,Z 232.551,A 10.516,B 90.000,C 0.000} C_DIS
LIN {X -285.166,Y -52.728,Z 232.338,A 10.476,B 90.000,C 0.000} C_DIS
LIN {X -285.182,Y -52.644,Z 232.117,A 10.459,B 90.000,C 0.000} C_DIS
LIN {X -285.219,Y -52.443,Z 231.904,A 10.419,B 90.000,C 0.000} C_DIS
LIN {X -285.234,Y -52.360,Z 231.684,A 10.402,B 90.000,C 0.000} C_DIS
LIN {X -285.271,Y -52.159,Z 231.466,A 10.362,B 90.000,C 0.000} C_DIS
LIN {X -285.278,Y -52.117,Z 231.345,A 10.353,B 90.000,C 0.000} C_DIS
LIN {X -285.282,Y -52.096,Z 231.254,A 10.349,B 90.000,C 0.000} C_DIS
LIN {X -285.301,Y -51.996,Z 231.178,A 10.329,B 90.000,C 0.000} C_DIS
LIN {X -285.304,Y -51.975,Z 231.087,A 10.325,B 90.000,C 0.000} C_DIS
LIN {X -285.312,Y -51.933,Z 230.966,A 10.316,B 90.000,C 0.000} C_DIS
LIN {X -285.348,Y -51.732,Z 230.748,A 10.276,B 90.000,C 0.000} C_DIS
LIN {X -285.364,Y -51.649,Z 230.528,A 10.259,B 90.000,C 0.000} C_DIS
LIN {X -285.400,Y -51.448,Z 230.314,A 10.219,B 90.000,C 0.000} C_DIS
LIN {X -285.415,Y -51.364,Z 230.094,A 10.202,B 90.000,C 0.000} C_DIS
LIN {X -285.451,Y -51.163,Z 229.881,A 10.162,B 90.000,C 0.000} C_DIS
LIN {X -285.466,Y -51.080,Z 229.661,A 10.145,B 90.000,C 0.000} C_DIS
LIN {X -285.502,Y -50.879,Z 229.447,A 10.105,B 90.000,C 0.000} C_DIS
LIN {X -285.517,Y -50.795,Z 229.227,A 10.088,B 90.000,C 0.000} C_DIS
LIN {X -285.552,Y -50.594,Z 229.009,A 10.047,B 90.000,C 0.000} C_DIS
LIN {X -285.560,Y -50.552,Z 228.888,A 10.039,B 90.000,C 0.000} C_DIS
LIN {X -285.564,Y -50.532,Z 228.797,A 10.035,B 90.000,C 0.000} C_DIS
LIN {X -285.581,Y -50.431,Z 228.721,A 10.015,B 90.000,C 0.000} C_DIS
LIN {X -285.585,Y -50.410,Z 228.630,A 10.010,B 90.000,C 0.000} C_DIS
LIN {X -285.592,Y -50.368,Z 228.509,A 10.002,B 90.000,C 0.000} C_DIS
LIN {X -285.628,Y -50.167,Z 228.291,A 9.962,B 90.000,C 0.000} C_DIS
LIN {X -285.642,Y -50.084,Z 228.071,A 9.945,B 90.000,C 0.000} C_DIS
LIN {X -285.678,Y -49.883,Z 227.857,A 9.905,B 90.000,C 0.000} C_DIS
LIN {X -285.692,Y -49.799,Z 227.637,A 9.888,B 90.000,C 0.000} C_DIS
LIN {X -285.727,Y -49.598,Z 227.424,A 9.848,B 90.000,C 0.000} C_DIS
LIN {X -285.742,Y -49.514,Z 227.204,A 9.831,B 90.000,C 0.000} C_DIS
LIN {X -285.777,Y -49.313,Z 226.986,A 9.790,B 90.000,C 0.000} C_DIS
LIN {X -285.784,Y -49.271,Z 226.864,A 9.782,B 90.000,C 0.000} C_DIS
LIN {X -285.787,Y -49.250,Z 226.773,A 9.778,B 90.000,C 0.000} C_DIS
LIN {X -285.805,Y -49.150,Z 226.698,A 9.758,B 90.000,C 0.000} C_DIS
LIN {X -285.808,Y -49.129,Z 226.607,A 9.753,B 90.000,C 0.000} C_DIS
LIN {X -285.815,Y -49.087,Z 226.486,A 9.745,B 90.000,C 0.000} C_DIS
LIN {X -285.850,Y -48.886,Z 226.268,A 9.705,B 90.000,C 0.000} C_DIS
LIN {X -285.864,Y -48.802,Z 226.047,A 9.688,B 90.000,C 0.000} C_DIS
LIN {X -285.899,Y -48.601,Z 225.829,A 9.648,B 90.000,C 0.000} C_DIS
LIN {X -285.906,Y -48.559,Z 225.708,A 9.639,B 90.000,C 0.000} C_DIS
LIN {X -285.914,Y -48.511,Z 225.608,A 9.630,B 90.000,C 0.000} C_DIS
LIN {X -285.942,Y -48.345,Z 225.579,A 9.596,B 90.000,C 0.000} C_DIS
LIN {X -285.967,Y -48.194,Z 225.601,A 9.566,B 90.000,C 0.000} C_DIS
LIN {X -285.978,Y -48.131,Z 225.652,A 9.554,B 90.000,C 0.000} C_DIS
LIN {X -285.992,Y -48.048,Z 225.703,A 9.537,B 90.000,C 0.000} C_DIS
LIN {X -286.026,Y -47.846,Z 225.724,A 9.496,B 90.000,C 0.000} C_DIS
LIN {X -286.059,Y -47.645,Z 225.703,A 9.456,B 90.000,C 0.000} C_DIS
LIN {X -286.073,Y -47.561,Z 225.652,A 9.439,B 90.000,C 0.000} C_DIS
LIN {X -286.079,Y -47.528,Z 225.601,A 9.433,B 90.000,C 0.000} C_DIS
LIN {X -286.110,Y -47.339,Z 225.550,A 9.395,B 90.000,C 0.000} C_DIS
LIN {X -286.127,Y -47.237,Z 225.474,A 9.375,B 90.000,C 0.000} C_DIS
LIN {X -286.139,Y -47.162,Z 225.371,A 9.360,B 90.000,C 0.000} C_DIS
LIN {X -286.148,Y -47.112,Z 225.179,A 9.350,B 90.000,C 0.000} C_DIS
LIN {X -286.156,Y -47.062,Z 225.146,A 9.339,B 90.000,C 0.000} C_DIS
LIN {X -286.164,Y -47.012,Z 225.040,A 9.329,B 90.000,C 0.000} C_DIS
LIN {X -286.171,Y -46.970,Z 224.529,A 9.321,B 90.000,C 0.000} C_DIS
LIN {X -286.179,Y -46.919,Z 224.423,A 9.311,B 90.000,C 0.000} C_DIS
LIN {X -286.188,Y -46.869,Z 224.279,A 9.301,B 90.000,C 0.000} C_DIS
LIN {X -286.194,Y -46.828,Z 223.556,A 9.293,B 90.000,C 0.000} C_DIS
LIN {X -286.203,Y -46.777,Z 223.411,A 9.282,B 90.000,C 0.000} C_DIS
LIN {X -286.211,Y -46.726,Z 223.310,A 9.272,B 90.000,C 0.000} C_DIS
LIN {X -286.219,Y -46.675,Z 222.773,A 9.262,B 90.000,C 0.000} C_DIS
LIN {X -286.237,Y -46.563,Z 222.617,A 9.239,B 90.000,C 0.000} C_DIS
LIN {X -286.254,Y -46.462,Z 222.505,A 9.219,B 90.000,C 0.000} C_DIS
LIN {X -286.261,Y -46.420,Z 222.384,A 9.211,B 90.000,C 0.000} C_DIS
LIN {X -286.264,Y -46.399,Z 222.293,A 9.207,B 90.000,C 0.000} C_DIS
LIN {X -286.280,Y -46.298,Z 222.217,A 9.187,B 90.000,C 0.000} C_DIS
LIN {X -286.284,Y -46.278,Z 222.127,A 9.182,B 90.000,C 0.000} C_DIS
LIN {X -286.291,Y -46.236,Z 222.005,A 9.174,B 90.000,C 0.000} C_DIS
LIN {X -286.323,Y -46.034,Z 221.787,A 9.134,B 90.000,C 0.000} C_DIS
LIN {X -286.336,Y -45.950,Z 221.567,A 9.117,B 90.000,C 0.000} C_DIS
LIN {X -286.369,Y -45.749,Z 221.354,A 9.077,B 90.000,C 0.000} C_DIS
LIN {X -286.382,Y -45.665,Z 221.133,A 9.060,B 90.000,C 0.000} C_DIS
LIN {X -286.414,Y -45.463,Z 220.920,A 9.019,B 90.000,C 0.000} C_DIS
LIN {X -286.428,Y -45.379,Z 220.700,A 9.003,B 90.000,C 0.000} C_DIS
LIN {X -286.459,Y -45.178,Z 220.482,A 8.962,B 90.000,C 0.000} C_DIS
LIN {X -286.466,Y -45.136,Z 220.360,A 8.954,B 90.000,C 0.000} C_DIS
LIN {X -286.469,Y -45.115,Z 220.270,A 8.950,B 90.000,C 0.000} C_DIS
LIN {X -286.485,Y -45.014,Z 220.194,A 8.930,B 90.000,C 0.000} C_DIS
LIN {X -286.488,Y -44.993,Z 220.103,A 8.925,B 90.000,C 0.000} C_DIS
LIN {X -286.495,Y -44.951,Z 219.982,A 8.917,B 90.000,C 0.000} C_DIS
LIN {X -286.527,Y -44.749,Z 219.764,A 8.877,B 90.000,C 0.000} C_DIS
LIN {X -286.540,Y -44.665,Z 219.544,A 8.860,B 90.000,C 0.000} C_DIS
LIN {X -286.571,Y -44.464,Z 219.330,A 8.820,B 90.000,C 0.000} C_DIS
LIN {X -286.584,Y -44.380,Z 219.110,A 8.803,B 90.000,C 0.000} C_DIS
LIN {X -286.615,Y -44.178,Z 218.897,A 8.762,B 90.000,C 0.000} C_DIS
LIN {X -286.628,Y -44.094,Z 218.676,A 8.746,B 90.000,C 0.000} C_DIS
LIN {X -286.659,Y -43.892,Z 218.463,A 8.705,B 90.000,C 0.000} C_DIS
LIN {X -286.672,Y -43.808,Z 218.243,A 8.689,B 90.000,C 0.000} C_DIS
LIN {X -286.703,Y -43.607,Z 218.025,A 8.648,B 90.000,C 0.000} C_DIS
LIN {X -286.709,Y -43.565,Z 217.903,A 8.640,B 90.000,C 0.000} C_DIS
LIN {X -286.712,Y -43.544,Z 217.813,A 8.636,B 90.000,C 0.000} C_DIS
LIN {X -286.728,Y -43.443,Z 217.737,A 8.615,B 90.000,C 0.000} C_DIS
LIN {X -286.731,Y -43.422,Z 217.646,A 8.611,B 90.000,C 0.000} C_DIS
LIN {X -286.737,Y -43.380,Z 217.525,A 8.603,B 90.000,C 0.000} C_DIS
LIN {X -286.768,Y -43.178,Z 217.307,A 8.563,B 90.000,C 0.000} C_DIS
LIN {X -286.780,Y -43.094,Z 217.087,A 8.546,B 90.000,C 0.000} C_DIS
LIN {X -286.811,Y -42.892,Z 216.873,A 8.505,B 90.000,C 0.000} C_DIS
LIN {X -286.823,Y -42.808,Z 216.653,A 8.489,B 90.000,C 0.000} C_DIS
LIN {X -286.853,Y -42.606,Z 216.440,A 8.448,B 90.000,C 0.000} C_DIS
LIN {X -286.866,Y -42.522,Z 216.219,A 8.432,B 90.000,C 0.000} C_DIS
LIN {X -286.895,Y -42.320,Z 216.001,A 8.391,B 90.000,C 0.000} C_DIS
LIN {X -286.902,Y -42.278,Z 215.880,A 8.383,B 90.000,C 0.000} C_DIS
LIN {X -286.905,Y -42.257,Z 215.789,A 8.379,B 90.000,C 0.000} C_DIS
LIN {X -286.920,Y -42.156,Z 215.714,A 8.358,B 90.000,C 0.000} C_DIS
LIN {X -286.923,Y -42.135,Z 215.623,A 8.354,B 90.000,C 0.000} C_DIS
LIN {X -286.929,Y -42.093,Z 215.501,A 8.346,B 90.000,C 0.000} C_DIS
LIN {X -286.958,Y -41.891,Z 215.283,A 8.306,B 90.000,C 0.000} C_DIS
LIN {X -286.971,Y -41.807,Z 215.063,A 8.289,B 90.000,C 0.000} C_DIS
LIN {X -287.000,Y -41.605,Z 214.850,A 8.248,B 90.000,C 0.000} C_DIS
LIN {X -287.012,Y -41.521,Z 214.630,A 8.232,B 90.000,C 0.000} C_DIS
LIN {X -287.041,Y -41.319,Z 214.416,A 8.191,B 90.000,C 0.000} C_DIS
LIN {X -287.053,Y -41.235,Z 214.196,A 8.175,B 90.000,C 0.000} C_DIS
LIN {X -287.082,Y -41.033,Z 213.983,A 8.134,B 90.000,C 0.000} C_DIS
LIN {X -287.094,Y -40.949,Z 213.762,A 8.117,B 90.000,C 0.000} C_DIS
LIN {X -287.123,Y -40.747,Z 213.544,A 8.077,B 90.000,C 0.000} C_DIS
LIN {X -287.129,Y -40.705,Z 213.423,A 8.069,B 90.000,C 0.000} C_DIS
LIN {X -287.132,Y -40.684,Z 213.332,A 8.065,B 90.000,C 0.000} C_DIS
LIN {X -287.146,Y -40.583,Z 213.257,A 8.044,B 90.000,C 0.000} C_DIS
LIN {X -287.149,Y -40.562,Z 213.166,A 8.040,B 90.000,C 0.000} C_DIS
LIN {X -287.155,Y -40.520,Z 213.044,A 8.032,B 90.000,C 0.000} C_DIS
LIN {X -287.184,Y -40.317,Z 212.826,A 7.991,B 90.000,C 0.000} C_DIS
LIN {X -287.196,Y -40.233,Z 212.606,A 7.975,B 90.000,C 0.000} C_DIS
LIN {X -287.224,Y -40.031,Z 212.393,A 7.934,B 90.000,C 0.000} C_DIS
LIN {X -287.235,Y -39.947,Z 212.173,A 7.918,B 90.000,C 0.000} C_DIS
LIN {X -287.264,Y -39.745,Z 211.959,A 7.877,B 90.000,C 0.000} C_DIS
LIN {X -287.275,Y -39.661,Z 211.739,A 7.860,B 90.000,C 0.000} C_DIS
LIN {X -287.303,Y -39.459,Z 211.521,A 7.820,B 90.000,C 0.000} C_DIS
LIN {X -287.309,Y -39.416,Z 211.400,A 7.812,B 90.000,C 0.000} C_DIS
LIN {X -287.312,Y -39.395,Z 211.309,A 7.808,B 90.000,C 0.000} C_DIS
LIN {X -287.326,Y -39.294,Z 211.233,A 7.787,B 90.000,C 0.000} C_DIS
LIN {X -287.328,Y -39.273,Z 211.142,A 7.783,B 90.000,C 0.000} C_DIS
LIN {X -287.334,Y -39.231,Z 211.021,A 7.775,B 90.000,C 0.000} C_DIS
LIN {X -287.362,Y -39.029,Z 210.803,A 7.734,B 90.000,C 0.000} C_DIS
LIN {X -287.373,Y -38.945,Z 210.583,A 7.718,B 90.000,C 0.000} C_DIS
LIN {X -287.400,Y -38.742,Z 210.369,A 7.677,B 90.000,C 0.000} C_DIS
LIN {X -287.412,Y -38.658,Z 210.149,A 7.661,B 90.000,C 0.000} C_DIS
LIN {X -287.439,Y -38.456,Z 209.936,A 7.620,B 90.000,C 0.000} C_DIS
LIN {X -287.450,Y -38.372,Z 209.716,A 7.603,B 90.000,C 0.000} C_DIS
LIN {X -287.477,Y -38.169,Z 209.498,A 7.563,B 90.000,C 0.000} C_DIS
LIN {X -287.483,Y -38.127,Z 209.376,A 7.555,B 90.000,C 0.000} C_DIS
LIN {X -287.485,Y -38.106,Z 209.285,A 7.551,B 90.000,C 0.000} C_DIS
LIN {X -287.499,Y -38.005,Z 209.210,A 7.530,B 90.000,C 0.000} C_DIS
LIN {X -287.502,Y -37.984,Z 209.119,A 7.526,B 90.000,C 0.000} C_DIS
LIN {X -287.507,Y -37.942,Z 208.998,A 7.518,B 90.000,C 0.000} C_DIS
LIN {X -287.534,Y -37.740,Z 208.780,A 7.477,B 90.000,C 0.000} C_DIS
LIN {X -287.545,Y -37.655,Z 208.559,A 7.461,B 90.000,C 0.000} C_DIS
LIN {X -287.571,Y -37.453,Z 208.346,A 7.420,B 90.000,C 0.000} C_DIS
LIN {X -287.582,Y -37.369,Z 208.126,A 7.404,B 90.000,C 0.000} C_DIS
LIN {X -287.609,Y -37.166,Z 207.913,A 7.363,B 90.000,C 0.000} C_DIS
LIN {X -287.619,Y -37.082,Z 207.692,A 7.346,B 90.000,C 0.000} C_DIS
LIN {X -287.645,Y -36.880,Z 207.479,A 7.306,B 90.000,C 0.000} C_DIS
LIN {X -287.656,Y -36.795,Z 207.259,A 7.289,B 90.000,C 0.000} C_DIS
LIN {X -287.682,Y -36.593,Z 207.041,A 7.249,B 90.000,C 0.000} C_DIS
LIN {X -287.687,Y -36.551,Z 206.919,A 7.241,B 90.000,C 0.000} C_DIS
LIN {X -287.690,Y -36.530,Z 206.828,A 7.236,B 90.000,C 0.000} C_DIS
LIN {X -287.703,Y -36.429,Z 206.753,A 7.216,B 90.000,C 0.000} C_DIS
LIN {X -287.706,Y -36.407,Z 206.662,A 7.212,B 90.000,C 0.000} C_DIS
LIN {X -287.711,Y -36.365,Z 206.541,A 7.204,B 90.000,C 0.000} C_DIS
LIN {X -287.736,Y -36.163,Z 206.323,A 7.163,B 90.000,C 0.000} C_DIS
LIN {X -287.747,Y -36.079,Z 206.102,A 7.147,B 90.000,C 0.000} C_DIS
LIN {X -287.772,Y -35.876,Z 205.889,A 7.106,B 90.000,C 0.000} C_DIS
LIN {X -287.783,Y -35.792,Z 205.669,A 7.090,B 90.000,C 0.000} C_DIS
LIN {X -287.808,Y -35.589,Z 205.456,A 7.049,B 90.000,C 0.000} C_DIS
LIN {X -287.818,Y -35.505,Z 205.235,A 7.032,B 90.000,C 0.000} C_DIS
LIN {X -287.843,Y -35.302,Z 205.017,A 6.992,B 90.000,C 0.000} C_DIS
LIN {X -287.848,Y -35.260,Z 204.896,A 6.984,B 90.000,C 0.000} C_DIS
LIN {X -287.851,Y -35.239,Z 204.805,A 6.979,B 90.000,C 0.000} C_DIS
LIN {X -287.863,Y -35.138,Z 204.729,A 6.959,B 90.000,C 0.000} C_DIS
LIN {X -287.866,Y -35.117,Z 204.639,A 6.955,B 90.000,C 0.000} C_DIS
LIN {X -287.871,Y -35.074,Z 204.517,A 6.947,B 90.000,C 0.000} C_DIS
LIN {X -287.896,Y -34.872,Z 204.299,A 6.906,B 90.000,C 0.000} C_DIS
LIN {X -287.906,Y -34.788,Z 204.079,A 6.890,B 90.000,C 0.000} C_DIS
LIN {X -287.930,Y -34.585,Z 203.866,A 6.849,B 90.000,C 0.000} C_DIS
LIN {X -287.940,Y -34.501,Z 203.645,A 6.833,B 90.000,C 0.000} C_DIS
LIN {X -287.965,Y -34.298,Z 203.432,A 6.792,B 90.000,C 0.000} C_DIS
LIN {X -287.975,Y -34.214,Z 203.212,A 6.775,B 90.000,C 0.000} C_DIS
LIN {X -287.999,Y -34.011,Z 202.999,A 6.735,B 90.000,C 0.000} C_DIS
LIN {X -288.009,Y -33.926,Z 202.778,A 6.718,B 90.000,C 0.000} C_DIS
LIN {X -288.032,Y -33.724,Z 202.560,A 6.678,B 90.000,C 0.000} C_DIS
LIN {X -288.037,Y -33.682,Z 202.439,A 6.670,B 90.000,C 0.000} C_DIS
LIN {X -288.040,Y -33.660,Z 202.348,A 6.665,B 90.000,C 0.000} C_DIS
LIN {X -288.052,Y -33.559,Z 202.273,A 6.645,B 90.000,C 0.000} C_DIS
LIN {X -288.054,Y -33.538,Z 202.182,A 6.641,B 90.000,C 0.000} C_DIS
LIN {X -288.059,Y -33.496,Z 202.060,A 6.633,B 90.000,C 0.000} C_DIS
LIN {X -288.083,Y -33.293,Z 201.842,A 6.592,B 90.000,C 0.000} C_DIS
LIN {X -288.092,Y -33.209,Z 201.622,A 6.576,B 90.000,C 0.000} C_DIS
LIN {X -288.116,Y -33.006,Z 201.409,A 6.535,B 90.000,C 0.000} C_DIS
LIN {X -288.125,Y -32.922,Z 201.188,A 6.518,B 90.000,C 0.000} C_DIS
LIN {X -288.148,Y -32.719,Z 200.975,A 6.478,B 90.000,C 0.000} C_DIS
LIN {X -288.158,Y -32.634,Z 200.755,A 6.461,B 90.000,C 0.000} C_DIS
LIN {X -288.181,Y -32.431,Z 200.537,A 6.421,B 90.000,C 0.000} C_DIS
LIN {X -288.186,Y -32.389,Z 200.415,A 6.413,B 90.000,C 0.000} C_DIS
LIN {X -288.188,Y -32.368,Z 200.325,A 6.408,B 90.000,C 0.000} C_DIS
LIN {X -288.199,Y -32.267,Z 200.249,A 6.388,B 90.000,C 0.000} C_DIS
LIN {X -288.202,Y -32.246,Z 200.158,A 6.384,B 90.000,C 0.000} C_DIS
LIN {X -288.206,Y -32.203,Z 200.037,A 6.376,B 90.000,C 0.000} C_DIS
LIN {X -288.229,Y -32.001,Z 199.819,A 6.335,B 90.000,C 0.000} C_DIS
LIN {X -288.238,Y -31.916,Z 199.599,A 6.319,B 90.000,C 0.000} C_DIS
LIN {X -288.261,Y -31.713,Z 199.385,A 6.278,B 90.000,C 0.000} C_DIS
LIN {X -288.270,Y -31.629,Z 199.165,A 6.261,B 90.000,C 0.000} C_DIS
LIN {X -288.292,Y -31.426,Z 198.952,A 6.221,B 90.000,C 0.000} C_DIS
LIN {X -288.301,Y -31.341,Z 198.731,A 6.204,B 90.000,C 0.000} C_DIS
LIN {X -288.323,Y -31.139,Z 198.513,A 6.164,B 90.000,C 0.000} C_DIS
LIN {X -288.328,Y -31.096,Z 198.392,A 6.156,B 90.000,C 0.000} C_DIS
LIN {X -288.330,Y -31.075,Z 198.301,A 6.151,B 90.000,C 0.000} C_DIS
LIN {X -288.341,Y -30.974,Z 198.226,A 6.131,B 90.000,C 0.000} C_DIS
LIN {X -288.343,Y -30.953,Z 198.135,A 6.127,B 90.000,C 0.000} C_DIS
LIN {X -288.348,Y -30.910,Z 198.014,A 6.119,B 90.000,C 0.000} C_DIS
LIN {X -288.370,Y -30.707,Z 197.796,A 6.078,B 90.000,C 0.000} C_DIS
LIN {X -288.379,Y -30.623,Z 197.575,A 6.062,B 90.000,C 0.000} C_DIS
LIN {X -288.400,Y -30.420,Z 197.362,A 6.021,B 90.000,C 0.000} C_DIS
LIN {X -288.409,Y -30.336,Z 197.142,A 6.004,B 90.000,C 0.000} C_DIS
LIN {X -288.430,Y -30.132,Z 196.928,A 5.964,B 90.000,C 0.000} C_DIS
LIN {X -288.439,Y -30.048,Z 196.708,A 5.947,B 90.000,C 0.000} C_DIS
LIN {X -288.460,Y -29.845,Z 196.495,A 5.907,B 90.000,C 0.000} C_DIS
LIN {X -288.469,Y -29.761,Z 196.274,A 5.890,B 90.000,C 0.000} C_DIS
LIN {X -288.490,Y -29.557,Z 196.057,A 5.850,B 90.000,C 0.000} C_DIS
LIN {X -288.494,Y -29.515,Z 195.935,A 5.841,B 90.000,C 0.000} C_DIS
LIN {X -288.496,Y -29.494,Z 195.844,A 5.837,B 90.000,C 0.000} C_DIS
LIN {X -288.507,Y -29.393,Z 195.769,A 5.817,B 90.000,C 0.000} C_DIS
LIN {X -288.509,Y -29.371,Z 195.678,A 5.813,B 90.000,C 0.000} C_DIS
LIN {X -288.513,Y -29.329,Z 195.557,A 5.805,B 90.000,C 0.000} C_DIS
LIN {X -288.534,Y -29.126,Z 195.339,A 5.764,B 90.000,C 0.000} C_DIS
LIN {X -288.542,Y -29.042,Z 195.118,A 5.747,B 90.000,C 0.000} C_DIS
LIN {X -288.563,Y -28.838,Z 194.905,A 5.707,B 90.000,C 0.000} C_DIS
LIN {X -288.571,Y -28.754,Z 194.685,A 5.690,B 90.000,C 0.000} C_DIS
LIN {X -288.591,Y -28.551,Z 194.471,A 5.650,B 90.000,C 0.000} C_DIS
LIN {X -288.599,Y -28.466,Z 194.251,A 5.633,B 90.000,C 0.000} C_DIS
LIN {X -288.619,Y -28.263,Z 194.033,A 5.593,B 90.000,C 0.000} C_DIS
LIN {X -288.624,Y -28.221,Z 193.912,A 5.584,B 90.000,C 0.000} C_DIS
LIN {X -288.626,Y -28.200,Z 193.821,A 5.580,B 90.000,C 0.000} C_DIS
LIN {X -288.636,Y -28.098,Z 193.745,A 5.560,B 90.000,C 0.000} C_DIS
LIN {X -288.638,Y -28.077,Z 193.655,A 5.556,B 90.000,C 0.000} C_DIS
LIN {X -288.642,Y -28.035,Z 193.533,A 5.548,B 90.000,C 0.000} C_DIS
LIN {X -288.661,Y -27.832,Z 193.315,A 5.507,B 90.000,C 0.000} C_DIS
LIN {X -288.670,Y -27.747,Z 193.095,A 5.490,B 90.000,C 0.000} C_DIS
LIN {X -288.689,Y -27.544,Z 192.882,A 5.450,B 90.000,C 0.000} C_DIS
LIN {X -288.697,Y -27.459,Z 192.661,A 5.433,B 90.000,C 0.000} C_DIS
LIN {X -288.714,Y -27.278,Z 192.464,A 5.397,B 90.000,C 0.000} C_DIS
LIN {X -288.718,Y -27.235,Z 192.265,A 5.389,B 90.000,C 0.000} C_DIS
LIN {X -288.720,Y -27.214,Z 189.765,A 5.385,B 90.000,C 0.000} C_DIS
LIN {X -288.720,Y -27.214,Z 189.736,A 5.385,B 90.000,C 0.000} C_DIS
LIN {X -288.741,Y -26.998,Z 189.736,A 5.342,B 90.000,C 0.000} C_DIS
LIN {X -288.755,Y -26.846,Z 189.758,A 5.312,B 90.000,C 0.000} C_DIS
LIN {X -288.761,Y -26.782,Z 189.809,A 5.299,B 90.000,C 0.000} C_DIS
LIN {X -288.777,Y -26.602,Z 189.861,A 5.263,B 90.000,C 0.000} C_DIS
LIN {X -288.862,Y -25.667,Z 189.861,A 5.078,B 90.000,C 0.000} C_DIS
LIN {X -288.878,Y -25.487,Z 189.809,A 5.042,B 90.000,C 0.000} C_DIS
LIN {X -288.881,Y -25.454,Z 189.758,A 5.035,B 90.000,C 0.000} C_DIS
LIN {X -288.898,Y -25.263,Z 189.707,A 4.998,B 90.000,C 0.000} C_DIS
LIN {X -288.907,Y -25.160,Z 189.631,A 4.977,B 90.000,C 0.000} C_DIS
LIN {X -288.913,Y -25.084,Z 189.528,A 4.962,B 90.000,C 0.000} C_DIS
LIN {X -288.917,Y -25.034,Z 189.336,A 4.952,B 90.000,C 0.000} C_DIS
LIN {X -288.922,Y -24.983,Z 189.303,A 4.942,B 90.000,C 0.000} C_DIS
LIN {X -288.926,Y -24.932,Z 189.197,A 4.932,B 90.000,C 0.000} C_DIS
LIN {X -288.928,Y -24.911,Z 188.942,A 4.928,B 90.000,C 0.000} C_DIS
LIN {X -288.926,Y -24.932,Z 188.686,A 4.932,B 90.000,C 0.000} C_DIS
LIN {X -288.917,Y -25.034,Z 188.474,A 4.952,B 90.000,C 0.000} C_DIS
LIN {X -288.914,Y -25.076,Z 187.964,A 4.961,B 90.000,C 0.000} C_DIS
LIN {X -288.909,Y -25.127,Z 187.858,A 4.971,B 90.000,C 0.000} C_DIS
LIN {X -288.905,Y -25.178,Z 187.794,A 4.981,B 90.000,C 0.000} C_DIS
LIN {X -288.901,Y -25.220,Z 187.488,A 4.989,B 90.000,C 0.000} C_DIS
LIN {X -288.897,Y -25.271,Z 187.424,A 4.999,B 90.000,C 0.000} C_DIS
LIN {X -288.892,Y -25.322,Z 187.339,A 5.009,B 90.000,C 0.000} C_DIS
LIN {X -288.889,Y -25.364,Z 186.931,A 5.018,B 90.000,C 0.000} C_DIS
LIN {X -288.880,Y -25.466,Z 186.761,A 5.038,B 90.000,C 0.000} C_DIS
LIN {X -288.876,Y -25.508,Z 186.353,A 5.046,B 90.000,C 0.000} C_DIS
LIN {X -288.867,Y -25.610,Z 186.183,A 5.066,B 90.000,C 0.000} C_DIS
LIN {X -288.863,Y -25.652,Z 185.775,A 5.075,B 90.000,C 0.000} C_DIS
LIN {X -288.854,Y -25.754,Z 185.605,A 5.095,B 90.000,C 0.000} C_DIS
LIN {X -288.850,Y -25.796,Z 185.196,A 5.103,B 90.000,C 0.000} C_DIS
LIN {X -288.841,Y -25.898,Z 185.027,A 5.123,B 90.000,C 0.000} C_DIS
LIN {X -288.838,Y -25.940,Z 184.618,A 5.132,B 90.000,C 0.000} C_DIS
LIN {X -288.828,Y -26.042,Z 184.449,A 5.152,B 90.000,C 0.000} C_DIS
LIN {X -288.825,Y -26.084,Z 184.040,A 5.160,B 90.000,C 0.000} C_DIS
LIN {X -288.815,Y -26.186,Z 183.870,A 5.181,B 90.000,C 0.000} C_DIS
LIN {X -288.812,Y -26.228,Z 183.462,A 5.189,B 90.000,C 0.000} C_DIS
LIN {X -288.802,Y -26.329,Z 183.292,A 5.209,B 90.000,C 0.000} C_DIS
LIN {X -288.798,Y -26.372,Z 182.884,A 5.218,B 90.000,C 0.000} C_DIS
LIN {X -288.794,Y -26.423,Z 182.799,A 5.228,B 90.000,C 0.000} C_DIS
LIN {X -288.789,Y -26.473,Z 182.735,A 5.238,B 90.000,C 0.000} C_DIS
LIN {X -288.785,Y -26.516,Z 182.429,A 5.246,B 90.000,C 0.000} C_DIS
LIN {X -288.781,Y -26.566,Z 182.365,A 5.256,B 90.000,C 0.000} C_DIS
LIN {X -288.776,Y -26.617,Z 182.281,A 5.266,B 90.000,C 0.000} C_DIS
LIN {X -288.772,Y -26.660,Z 181.872,A 5.275,B 90.000,C 0.000} C_DIS
LIN {X -288.763,Y -26.761,Z 181.702,A 5.295,B 90.000,C 0.000} C_DIS
LIN {X -288.759,Y -26.803,Z 181.294,A 5.303,B 90.000,C 0.000} C_DIS
LIN {X -288.749,Y -26.905,Z 181.124,A 5.323,B 90.000,C 0.000} C_DIS
LIN {X -288.745,Y -26.947,Z 180.716,A 5.332,B 90.000,C 0.000} C_DIS
LIN {X -288.741,Y -26.998,Z 180.631,A 5.342,B 90.000,C 0.000} C_DIS
LIN {X -288.736,Y -27.051,Z 178.132,A 5.352,B 90.000,C 0.000} C_DIS
LIN {X -288.735,Y -27.058,Z 175.632,A 5.354,B 90.000,C 0.000} C_DIS
LIN {X -288.734,Y -27.064,Z 173.132,A 5.355,B 90.000,C 0.000} C_DIS
LIN {X -288.734,Y -27.070,Z 170.632,A 5.356,B 90.000,C 0.000} C_DIS
LIN {X -288.734,Y -27.064,Z 168.132,A 5.355,B 90.000,C 0.000} C_DIS
LIN {X -288.735,Y -27.058,Z 165.632,A 5.354,B 90.000,C 0.000} C_DIS
LIN {X -288.735,Y -27.053,Z 163.132,A 5.353,B 90.000,C 0.000} C_DIS
LIN {X -288.740,Y -27.003,Z 160.633,A 5.343,B 90.000,C 0.000} C_DIS
LIN {X -288.746,Y -26.935,Z 158.134,A 5.329,B 90.000,C 0.000} C_DIS
LIN {X -288.747,Y -26.926,Z 155.634,A 5.328,B 90.000,C 0.000} C_DIS
LIN {X -288.747,Y -26.926,Z 153.460,A 5.328,B 90.000,C 0.000} C_DIS
LIN {X -288.793,Y -26.435,Z 153.481,A 5.230,B 90.000,C 0.000} C_DIS
LIN {X -288.800,Y -26.350,Z 153.532,A 5.213,B 90.000,C 0.000} C_DIS
LIN {X -288.817,Y -26.170,Z 153.584,A 5.178,B 90.000,C 0.000} C_DIS
LIN {X -288.900,Y -25.235,Z 153.624,A 4.992,B 90.000,C 0.000} C_DIS
LIN {X -288.931,Y -24.875,Z 153.729,A 4.921,B 90.000,C 0.000} C_DIS
LIN {X -289.010,Y -23.939,Z 153.769,A 4.735,B 90.000,C 0.000} C_DIS
LIN {X -289.040,Y -23.578,Z 153.873,A 4.664,B 90.000,C 0.000} C_DIS
LIN {X -289.115,Y -22.642,Z 153.913,A 4.478,B 90.000,C 0.000} C_DIS
LIN {X -289.144,Y -22.264,Z 154.018,A 4.403,B 90.000,C 0.000} C_DIS
LIN {X -289.223,Y -21.219,Z 154.058,A 4.196,B 90.000,C 0.000} C_DIS
LIN {X -289.237,Y -21.021,Z 154.110,A 4.157,B 90.000,C 0.000} C_DIS
LIN {X -289.246,Y -20.895,Z 154.161,A 4.132,B 90.000,C 0.000} C_DIS
LIN {X -289.299,Y -20.156,Z 154.182,A 3.985,B 90.000,C 0.000} C_DIS
LIN {X -289.299,Y -20.156,Z 155.483,A 3.985,B 90.000,C 0.000} C_DIS
LIN {X -289.366,Y -19.164,Z 155.504,A 3.789,B 90.000,C 0.000} C_DIS
LIN {X -289.387,Y -18.840,Z 155.607,A 3.725,B 90.000,C 0.000} C_DIS
LIN {X -289.440,Y -18.011,Z 155.648,A 3.561,B 90.000,C 0.000} C_DIS
LIN {X -289.460,Y -17.686,Z 155.752,A 3.496,B 90.000,C 0.000} C_DIS
LIN {X -289.510,Y -16.857,Z 155.793,A 3.332,B 90.000,C 0.000} C_DIS
LIN {X -289.528,Y -16.532,Z 155.896,A 3.268,B 90.000,C 0.000} C_DIS
LIN {X -289.575,Y -15.702,Z 155.937,A 3.104,B 90.000,C 0.000} C_DIS
LIN {X -289.592,Y -15.386,Z 156.041,A 3.041,B 90.000,C 0.000} C_DIS
LIN {X -289.637,Y -14.512,Z 156.091,A 2.868,B 90.000,C 0.000} C_DIS
LIN {X -289.643,Y -14.385,Z 156.145,A 2.843,B 90.000,C 0.000} C_DIS
LIN {X -289.649,Y -14.274,Z 156.239,A 2.821,B 90.000,C 0.000} C_DIS
LIN {X -289.655,Y -14.148,Z 156.397,A 2.796,B 90.000,C 0.000} C_DIS
LIN {X -289.657,Y -14.096,Z 156.528,A 2.786,B 90.000,C 0.000} C_DIS
LIN {X -289.658,Y -14.075,Z 156.607,A 2.782,B 90.000,C 0.000} C_DIS
LIN {X -289.661,Y -14.024,Z 156.639,A 2.772,B 90.000,C 0.000} C_DIS
LIN {X -289.663,Y -13.973,Z 156.682,A 2.762,B 90.000,C 0.000} C_DIS
LIN {X -289.665,Y -13.931,Z 156.886,A 2.753,B 90.000,C 0.000} C_DIS
LIN {X -289.670,Y -13.829,Z 156.966,A 2.733,B 90.000,C 0.000} C_DIS
LIN {X -289.671,Y -13.808,Z 157.057,A 2.729,B 90.000,C 0.000} C_DIS
LIN {X -289.673,Y -13.765,Z 157.178,A 2.721,B 90.000,C 0.000} C_DIS
LIN {X -289.683,Y -13.561,Z 157.396,A 2.680,B 90.000,C 0.000} C_DIS
LIN {X -289.687,Y -13.476,Z 157.617,A 2.664,B 90.000,C 0.000} C_DIS
LIN {X -289.696,Y -13.273,Z 157.835,A 2.623,B 90.000,C 0.000} C_DIS
LIN {X -289.698,Y -13.230,Z 157.956,A 2.615,B 90.000,C 0.000} C_DIS
LIN {X -289.699,Y -13.209,Z 158.047,A 2.611,B 90.000,C 0.000} C_DIS
LIN {X -289.704,Y -13.107,Z 158.119,A 2.590,B 90.000,C 0.000} C_DIS
LIN {X -289.705,Y -13.086,Z 158.200,A 2.586,B 90.000,C 0.000} C_DIS
LIN {X -289.707,Y -13.022,Z 158.341,A 2.574,B 90.000,C 0.000} C_DIS
LIN {X -289.775,Y -11.406,Z 160.247,A 2.254,B 90.000,C 0.000} C_DIS
LIN {X -289.841,Y -9.594,Z 161.968,A 1.896,B 90.000,C 0.000} C_DIS
LIN {X -289.869,Y -8.721,Z 162.646,A 1.723,B 90.000,C 0.000} C_DIS
LIN {X -289.873,Y -8.580,Z 162.710,A 1.695,B 90.000,C 0.000} C_DIS
LIN {X -289.875,Y -8.498,Z 162.731,A 1.679,B 90.000,C 0.000} C_DIS
LIN {X -289.878,Y -8.426,Z 162.833,A 1.665,B 90.000,C 0.000} C_DIS
LIN {X -289.880,Y -8.336,Z 162.854,A 1.647,B 90.000,C 0.000} C_DIS
LIN {X -289.884,Y -8.214,Z 162.897,A 1.623,B 90.000,C 0.000} C_DIS
LIN {X -289.890,Y -7.992,Z 163.101,A 1.579,B 90.000,C 0.000} C_DIS
LIN {X -289.893,Y -7.870,Z 163.143,A 1.555,B 90.000,C 0.000} C_DIS
LIN {X -289.896,Y -7.780,Z 163.164,A 1.537,B 90.000,C 0.000} C_DIS
LIN {X -289.898,Y -7.699,Z 163.267,A 1.521,B 90.000,C 0.000} C_DIS
LIN {X -289.903,Y -7.495,Z 163.309,A 1.481,B 90.000,C 0.000} C_DIS
LIN {X -289.905,Y -7.410,Z 163.411,A 1.464,B 90.000,C 0.000} C_DIS
LIN {X -289.910,Y -7.206,Z 163.454,A 1.424,B 90.000,C 0.000} C_DIS
LIN {X -289.913,Y -7.121,Z 163.556,A 1.407,B 90.000,C 0.000} C_DIS
LIN {X -289.917,Y -6.917,Z 163.598,A 1.367,B 90.000,C 0.000} C_DIS
LIN {X -289.920,Y -6.832,Z 163.700,A 1.350,B 90.000,C 0.000} C_DIS
LIN {X -289.924,Y -6.628,Z 163.743,A 1.310,B 90.000,C 0.000} C_DIS
LIN {X -289.926,Y -6.543,Z 163.845,A 1.293,B 90.000,C 0.000} C_DIS
LIN {X -289.931,Y -6.339,Z 163.887,A 1.253,B 90.000,C 0.000} C_DIS
LIN {X -289.932,Y -6.297,Z 163.938,A 1.244,B 90.000,C 0.000} C_DIS
LIN {X -289.933,Y -6.233,Z 163.989,A 1.232,B 90.000,C 0.000} C_DIS
LIN {X -289.939,Y -5.927,Z 164.032,A 1.171,B 90.000,C 0.000} C_DIS
LIN {X -289.942,Y -5.800,Z 164.134,A 1.146,B 90.000,C 0.000} C_DIS
LIN {X -289.948,Y -5.494,Z 164.176,A 1.085,B 90.000,C 0.000} C_DIS
LIN {X -289.950,Y -5.366,Z 164.278,A 1.060,B 90.000,C 0.000} C_DIS
LIN {X -289.956,Y -5.060,Z 164.321,A 1.000,B 90.000,C 0.000} C_DIS
LIN {X -289.958,Y -4.933,Z 164.423,A 0.975,B 90.000,C 0.000} C_DIS
LIN {X -289.963,Y -4.627,Z 164.465,A 0.914,B 90.000,C 0.000} C_DIS
LIN {X -289.964,Y -4.563,Z 164.516,A 0.902,B 90.000,C 0.000} C_DIS
LIN {X -289.965,Y -4.478,Z 164.567,A 0.885,B 90.000,C 0.000} C_DIS
LIN {X -289.971,Y -4.070,Z 164.610,A 0.804,B 90.000,C 0.000} C_DIS
LIN {X -289.974,Y -3.879,Z 164.712,A 0.766,B 90.000,C 0.000} C_DIS
LIN {X -289.980,Y -3.368,Z 164.754,A 0.666,B 90.000,C 0.000} C_DIS
LIN {X -289.982,Y -3.262,Z 164.805,A 0.645,B 90.000,C 0.000} C_DIS
LIN {X -289.983,Y -3.118,Z 164.857,A 0.616,B 90.000,C 0.000} C_DIS
LIN {X -289.990,Y -2.395,Z 164.898,A 0.473,B 90.000,C 0.000} C_DIS
LIN {X -289.991,Y -2.251,Z 164.950,A 0.445,B 90.000,C 0.000} C_DIS
LIN {X -289.999,Y 0.249,Z 165.014,A -0.049,B 90.000,C 0.000} C_DIS
LIN {X -289.996,Y 1.507,Z 164.950,A -0.298,B 90.000,C 0.000} C_DIS
LIN {X -289.995,Y 1.652,Z 164.898,A -0.326,B 90.000,C 0.000} C_DIS
LIN {X -289.990,Y 2.374,Z 164.857,A -0.469,B 90.000,C 0.000} C_DIS
LIN {X -289.989,Y 2.519,Z 164.805,A -0.498,B 90.000,C 0.000} C_DIS
LIN {X -289.988,Y 2.625,Z 164.754,A -0.519,B 90.000,C 0.000} C_DIS
LIN {X -289.983,Y 3.135,Z 164.712,A -0.619,B 90.000,C 0.000} C_DIS
LIN {X -289.981,Y 3.326,Z 164.610,A -0.657,B 90.000,C 0.000} C_DIS
LIN {X -289.976,Y 3.735,Z 164.567,A -0.738,B 90.000,C 0.000} C_DIS
LIN {X -289.974,Y 3.904,Z 164.465,A -0.771,B 90.000,C 0.000} C_DIS
LIN {X -289.968,Y 4.313,Z 164.423,A -0.852,B 90.000,C 0.000} C_DIS
LIN {X -289.967,Y 4.398,Z 164.372,A -0.869,B 90.000,C 0.000} C_DIS
LIN {X -289.966,Y 4.461,Z 164.321,A -0.881,B 90.000,C 0.000} C_DIS
LIN {X -289.961,Y 4.767,Z 164.278,A -0.942,B 90.000,C 0.000} C_DIS
LIN {X -289.959,Y 4.895,Z 164.176,A -0.967,B 90.000,C 0.000} C_DIS
LIN {X -289.953,Y 5.201,Z 164.134,A -1.028,B 90.000,C 0.000} C_DIS
LIN {X -289.952,Y 5.265,Z 164.083,A -1.040,B 90.000,C 0.000} C_DIS
LIN {X -289.951,Y 5.307,Z 164.032,A -1.049,B 90.000,C 0.000} C_DIS
LIN {X -289.948,Y 5.511,Z 163.989,A -1.089,B 90.000,C 0.000} C_DIS
LIN {X -289.947,Y 5.554,Z 163.938,A -1.097,B 90.000,C 0.000} C_DIS
LIN {X -289.946,Y 5.617,Z 163.887,A -1.110,B 90.000,C 0.000} C_DIS
LIN {X -289.939,Y 5.923,Z 163.845,A -1.170,B 90.000,C 0.000} C_DIS
LIN {X -289.938,Y 5.987,Z 163.794,A -1.183,B 90.000,C 0.000} C_DIS
LIN {X -289.937,Y 6.030,Z 163.743,A -1.191,B 90.000,C 0.000} C_DIS
LIN {X -289.933,Y 6.234,Z 163.700,A -1.232,B 90.000,C 0.000} C_DIS
LIN {X -289.931,Y 6.319,Z 163.598,A -1.248,B 90.000,C 0.000} C_DIS
LIN {X -289.927,Y 6.523,Z 163.556,A -1.289,B 90.000,C 0.000} C_DIS
LIN {X -289.925,Y 6.607,Z 163.454,A -1.306,B 90.000,C 0.000} C_DIS
LIN {X -289.920,Y 6.812,Z 163.411,A -1.346,B 90.000,C 0.000} C_DIS
LIN {X -289.918,Y 6.896,Z 163.309,A -1.363,B 90.000,C 0.000} C_DIS
LIN {X -289.913,Y 7.101,Z 163.267,A -1.403,B 90.000,C 0.000} C_DIS
LIN {X -289.911,Y 7.181,Z 163.164,A -1.419,B 90.000,C 0.000} C_DIS
LIN {X -289.909,Y 7.272,Z 163.143,A -1.437,B 90.000,C 0.000} C_DIS
LIN {X -289.906,Y 7.393,Z 163.101,A -1.461,B 90.000,C 0.000} C_DIS
LIN {X -289.900,Y 7.616,Z 162.897,A -1.505,B 90.000,C 0.000} C_DIS
LIN {X -289.897,Y 7.737,Z 162.854,A -1.529,B 90.000,C 0.000} C_DIS
LIN {X -289.894,Y 7.828,Z 162.833,A -1.547,B 90.000,C 0.000} C_DIS
LIN {X -289.892,Y 7.899,Z 162.731,A -1.561,B 90.000,C 0.000} C_DIS
LIN {X -289.890,Y 7.981,Z 162.710,A -1.577,B 90.000,C 0.000} C_DIS
LIN {X -289.886,Y 8.122,Z 162.646,A -1.605,B 90.000,C 0.000} C_DIS
LIN {X -289.826,Y 10.037,Z 161.040,A -1.983,B 90.000,C 0.000} C_DIS
LIN {X -289.765,Y 11.660,Z 159.140,A -2.304,B 90.000,C 0.000} C_DIS
LIN {X -289.758,Y 11.846,Z 158.919,A -2.341,B 90.000,C 0.000} C_DIS
LIN {X -289.755,Y 11.910,Z 158.778,A -2.354,B 90.000,C 0.000} C_DIS
LIN {X -289.754,Y 11.931,Z 158.697,A -2.358,B 90.000,C 0.000} C_DIS
LIN {X -289.750,Y 12.033,Z 158.625,A -2.378,B 90.000,C 0.000} C_DIS
LIN {X -289.749,Y 12.054,Z 158.534,A -2.382,B 90.000,C 0.000} C_DIS
LIN {X -289.748,Y 12.097,Z 158.413,A -2.391,B 90.000,C 0.000} C_DIS
LIN {X -289.739,Y 12.301,Z 158.190,A -2.431,B 90.000,C 0.000} C_DIS
LIN {X -289.737,Y 12.343,Z 158.069,A -2.439,B 90.000,C 0.000} C_DIS
LIN {X -289.736,Y 12.364,Z 157.978,A -2.444,B 90.000,C 0.000} C_DIS
LIN {X -289.732,Y 12.466,Z 157.898,A -2.464,B 90.000,C 0.000} C_DIS
LIN {X -289.730,Y 12.509,Z 157.694,A -2.472,B 90.000,C 0.000} C_DIS
LIN {X -289.726,Y 12.611,Z 157.609,A -2.492,B 90.000,C 0.000} C_DIS
LIN {X -289.724,Y 12.653,Z 157.405,A -2.501,B 90.000,C 0.000} C_DIS
LIN {X -289.719,Y 12.755,Z 157.320,A -2.521,B 90.000,C 0.000} C_DIS
LIN {X -289.717,Y 12.797,Z 157.115,A -2.529,B 90.000,C 0.000} C_DIS
LIN {X -289.713,Y 12.899,Z 157.031,A -2.549,B 90.000,C 0.000} C_DIS
LIN {X -289.711,Y 12.942,Z 156.826,A -2.558,B 90.000,C 0.000} C_DIS
LIN {X -289.707,Y 13.044,Z 156.742,A -2.578,B 90.000,C 0.000} C_DIS
LIN {X -289.705,Y 13.086,Z 156.537,A -2.586,B 90.000,C 0.000} C_DIS
LIN {X -289.700,Y 13.188,Z 156.452,A -2.607,B 90.000,C 0.000} C_DIS
LIN {X -289.699,Y 13.209,Z 156.350,A -2.611,B 90.000,C 0.000} C_DIS
LIN {X -289.697,Y 13.245,Z 156.242,A -2.618,B 90.000,C 0.000} C_DIS
LIN {X -289.692,Y 13.354,Z 156.206,A -2.639,B 90.000,C 0.000} C_DIS
LIN {X -289.688,Y 13.456,Z 156.185,A -2.659,B 90.000,C 0.000} C_DIS
LIN {X -289.686,Y 13.498,Z 156.134,A -2.668,B 90.000,C 0.000} C_DIS
LIN {X -289.679,Y 13.642,Z 156.082,A -2.696,B 90.000,C 0.000} C_DIS
LIN {X -289.644,Y 14.364,Z 156.041,A -2.839,B 90.000,C 0.000} C_DIS
LIN {X -289.629,Y 14.671,Z 155.937,A -2.900,B 90.000,C 0.000} C_DIS
LIN {X -289.585,Y 15.501,Z 155.896,A -3.064,B 90.000,C 0.000} C_DIS
LIN {X -289.567,Y 15.844,Z 155.792,A -3.132,B 90.000,C 0.000} C_DIS
LIN {X -289.514,Y 16.782,Z 155.752,A -3.317,B 90.000,C 0.000} C_DIS
LIN {X -289.493,Y 17.142,Z 155.648,A -3.389,B 90.000,C 0.000} C_DIS
LIN {X -289.436,Y 18.080,Z 155.608,A -3.574,B 90.000,C 0.000} C_DIS
LIN {X -289.411,Y 18.469,Z 155.503,A -3.651,B 90.000,C 0.000} C_DIS
LIN {X -289.334,Y 19.638,Z 155.460,A -3.883,B 90.000,C 0.000} C_DIS
LIN {X -289.317,Y 19.888,Z 155.380,A -3.932,B 90.000,C 0.000} C_DIS
LIN {X -289.312,Y 19.961,Z 155.255,A -3.947,B 90.000,C 0.000} C_DIS
LIN {X -289.310,Y 19.988,Z 155.101,A -3.952,B 90.000,C 0.000} C_DIS
LIN {X -289.312,Y 19.968,Z 154.960,A -3.948,B 90.000,C 0.000} C_DIS
LIN {X -289.316,Y 19.901,Z 154.875,A -3.935,B 90.000,C 0.000} C_DIS
LIN {X -289.320,Y 19.847,Z 154.833,A -3.924,B 90.000,C 0.000} C_DIS
LIN {X -289.316,Y 19.901,Z 154.791,A -3.935,B 90.000,C 0.000} C_DIS
LIN {X -289.312,Y 19.964,Z 154.678,A -3.948,B 90.000,C 0.000} C_DIS
LIN {X -289.310,Y 19.991,Z 154.466,A -3.953,B 90.000,C 0.000} C_DIS
LIN {X -289.310,Y 19.991,Z 154.182,A -3.953,B 90.000,C 0.000} C_DIS
LIN {X -289.249,Y 20.856,Z 154.162,A -4.124,B 90.000,C 0.000} C_DIS
LIN {X -289.227,Y 21.162,Z 154.058,A -4.185,B 90.000,C 0.000} C_DIS
LIN {X -289.165,Y 21.991,Z 154.018,A -4.349,B 90.000,C 0.000} C_DIS
LIN {X -289.139,Y 22.333,Z 153.913,A -4.417,B 90.000,C 0.000} C_DIS
LIN {X -289.065,Y 23.270,Z 153.873,A -4.602,B 90.000,C 0.000} C_DIS
LIN {X -289.036,Y 23.630,Z 153.769,A -4.674,B 90.000,C 0.000} C_DIS
LIN {X -288.958,Y 24.566,Z 153.729,A -4.859,B 90.000,C 0.000} C_DIS
LIN {X -288.928,Y 24.908,Z 153.625,A -4.927,B 90.000,C 0.000} C_DIS
LIN {X -288.856,Y 25.736,Z 153.584,A -5.091,B 90.000,C 0.000} C_DIS
LIN {X -288.827,Y 26.060,Z 153.480,A -5.156,B 90.000,C 0.000} C_DIS
LIN {X -288.736,Y 27.049,Z 153.460,A -5.352,B 90.000,C 0.000} C_DIS
LIN {X -288.736,Y 27.049,Z 155.960,A -5.352,B 90.000,C 0.000} C_DIS
LIN {X -288.734,Y 27.063,Z 158.460,A -5.355,B 90.000,C 0.000} C_DIS
LIN {X -288.727,Y 27.144,Z 160.958,A -5.371,B 90.000,C 0.000} C_DIS
LIN {X -288.724,Y 27.177,Z 163.458,A -5.377,B 90.000,C 0.000} C_DIS
LIN {X -288.723,Y 27.183,Z 165.958,A -5.378,B 90.000,C 0.000} C_DIS
LIN {X -288.723,Y 27.188,Z 168.458,A -5.380,B 90.000,C 0.000} C_DIS
LIN {X -288.722,Y 27.192,Z 170.958,A -5.380,B 90.000,C 0.000} C_DIS
LIN {X -288.723,Y 27.187,Z 173.458,A -5.379,B 90.000,C 0.000} C_DIS
LIN {X -288.723,Y 27.181,Z 175.958,A -5.378,B 90.000,C 0.000} C_DIS
LIN {X -288.724,Y 27.175,Z 178.457,A -5.377,B 90.000,C 0.000} C_DIS
LIN {X -288.728,Y 27.129,Z 180.957,A -5.368,B 90.000,C 0.000} C_DIS
LIN {X -288.729,Y 27.121,Z 181.354,A -5.366,B 90.000,C 0.000} C_DIS
LIN {X -288.734,Y 27.070,Z 181.439,A -5.356,B 90.000,C 0.000} C_DIS
LIN {X -288.738,Y 27.028,Z 181.847,A -5.348,B 90.000,C 0.000} C_DIS
LIN {X -288.747,Y 26.926,Z 182.017,A -5.328,B 90.000,C 0.000} C_DIS
LIN {X -288.751,Y 26.884,Z 182.425,A -5.319,B 90.000,C 0.000} C_DIS
LIN {X -288.761,Y 26.782,Z 182.595,A -5.299,B 90.000,C 0.000} C_DIS
LIN {X -288.765,Y 26.740,Z 183.003,A -5.291,B 90.000,C 0.000} C_DIS
LIN {X -288.774,Y 26.638,Z 183.173,A -5.270,B 90.000,C 0.000} C_DIS
LIN {X -288.778,Y 26.596,Z 183.581,A -5.262,B 90.000,C 0.000} C_DIS
LIN {X -288.787,Y 26.495,Z 183.751,A -5.242,B 90.000,C 0.000} C_DIS
LIN {X -288.791,Y 26.452,Z 184.159,A -5.233,B 90.000,C 0.000} C_DIS
LIN {X -288.800,Y 26.351,Z 184.329,A -5.213,B 90.000,C 0.000} C_DIS
LIN {X -288.804,Y 26.308,Z 184.738,A -5.205,B 90.000,C 0.000} C_DIS
LIN {X -288.813,Y 26.207,Z 184.907,A -5.185,B 90.000,C 0.000} C_DIS
LIN {X -288.817,Y 26.164,Z 185.316,A -5.176,B 90.000,C 0.000} C_DIS
LIN {X -288.826,Y 26.063,Z 185.485,A -5.156,B 90.000,C 0.000} C_DIS
LIN {X -288.830,Y 26.020,Z 185.894,A -5.148,B 90.000,C 0.000} C_DIS
LIN {X -288.835,Y 25.970,Z 185.979,A -5.138,B 90.000,C 0.000} C_DIS
LIN {X -288.839,Y 25.919,Z 186.042,A -5.128,B 90.000,C 0.000} C_DIS
LIN {X -288.843,Y 25.877,Z 186.349,A -5.119,B 90.000,C 0.000} C_DIS
LIN {X -288.848,Y 25.826,Z 186.412,A -5.109,B 90.000,C 0.000} C_DIS
LIN {X -288.852,Y 25.775,Z 186.497,A -5.099,B 90.000,C 0.000} C_DIS
LIN {X -288.856,Y 25.733,Z 186.905,A -5.091,B 90.000,C 0.000} C_DIS
LIN {X -288.865,Y 25.631,Z 187.075,A -5.071,B 90.000,C 0.000} C_DIS
LIN {X -288.869,Y 25.589,Z 187.484,A -5.062,B 90.000,C 0.000} C_DIS
LIN {X -288.873,Y 25.538,Z 187.568,A -5.052,B 90.000,C 0.000} C_DIS
LIN {X -288.878,Y 25.487,Z 187.686,A -5.042,B 90.000,C 0.000} C_DIS
LIN {X -288.880,Y 25.466,Z 187.969,A -5.038,B 90.000,C 0.000} C_DIS
LIN {X -288.877,Y 25.500,Z 188.327,A -5.045,B 90.000,C 0.000} C_DIS
LIN {X -288.864,Y 25.642,Z 188.547,A -5.073,B 90.000,C 0.000} C_DIS
LIN {X -288.848,Y 25.821,Z 188.673,A -5.108,B 90.000,C 0.000} C_DIS
LIN {X -288.832,Y 26.002,Z 188.725,A -5.144,B 90.000,C 0.000} C_DIS
LIN {X -288.820,Y 26.132,Z 188.746,A -5.170,B 90.000,C 0.000} C_DIS
LIN {X -288.815,Y 26.186,Z 188.797,A -5.181,B 90.000,C 0.000} C_DIS
LIN {X -288.806,Y 26.291,Z 188.848,A -5.202,B 90.000,C 0.000} C_DIS
LIN {X -288.759,Y 26.799,Z 188.890,A -5.302,B 90.000,C 0.000} C_DIS
LIN {X -288.749,Y 26.905,Z 188.942,A -5.323,B 90.000,C 0.000} C_DIS
LIN {X -288.743,Y 26.969,Z 188.993,A -5.336,B 90.000,C 0.000} C_DIS
LIN {X -288.729,Y 27.121,Z 189.014,A -5.366,B 90.000,C 0.000} C_DIS
LIN {X -288.709,Y 27.337,Z 189.014,A -5.409,B 90.000,C 0.000} C_DIS
LIN {X -288.708,Y 27.348,Z 191.514,A -5.411,B 90.000,C 0.000} C_DIS
LIN {X -288.707,Y 27.358,Z 192.219,A -5.413,B 90.000,C 0.000} C_DIS
LIN {X -288.703,Y 27.401,Z 192.458,A -5.422,B 90.000,C 0.000} C_DIS
LIN {X -288.685,Y 27.583,Z 192.666,A -5.458,B 90.000,C 0.000} C_DIS
LIN {X -288.681,Y 27.625,Z 192.787,A -5.466,B 90.000,C 0.000} C_DIS
LIN {X -288.679,Y 27.646,Z 192.878,A -5.470,B 90.000,C 0.000} C_DIS
LIN {X -288.669,Y 27.748,Z 192.954,A -5.491,B 90.000,C 0.000} C_DIS
LIN {X -288.667,Y 27.769,Z 193.044,A -5.495,B 90.000,C 0.000} C_DIS
LIN {X -288.663,Y 27.811,Z 193.166,A -5.503,B 90.000,C 0.000} C_DIS
LIN {X -288.644,Y 28.014,Z 193.384,A -5.543,B 90.000,C 0.000} C_DIS
LIN {X -288.636,Y 28.099,Z 193.604,A -5.560,B 90.000,C 0.000} C_DIS
LIN {X -288.616,Y 28.302,Z 193.817,A -5.601,B 90.000,C 0.000} C_DIS
LIN {X -288.607,Y 28.386,Z 194.038,A -5.617,B 90.000,C 0.000} C_DIS
LIN {X -288.587,Y 28.589,Z 194.256,A -5.658,B 90.000,C 0.000} C_DIS
LIN {X -288.583,Y 28.632,Z 194.377,A -5.666,B 90.000,C 0.000} C_DIS
LIN {X -288.581,Y 28.653,Z 194.468,A -5.670,B 90.000,C 0.000} C_DIS
LIN {X -288.571,Y 28.754,Z 194.543,A -5.690,B 90.000,C 0.000} C_DIS
LIN {X -288.569,Y 28.776,Z 194.634,A -5.695,B 90.000,C 0.000} C_DIS
LIN {X -288.565,Y 28.818,Z 194.756,A -5.703,B 90.000,C 0.000} C_DIS
LIN {X -288.544,Y 29.021,Z 194.974,A -5.743,B 90.000,C 0.000} C_DIS
LIN {X -288.536,Y 29.105,Z 195.194,A -5.760,B 90.000,C 0.000} C_DIS
LIN {X -288.515,Y 29.308,Z 195.412,A -5.800,B 90.000,C 0.000} C_DIS
LIN {X -288.511,Y 29.351,Z 195.533,A -5.809,B 90.000,C 0.000} C_DIS
LIN {X -288.509,Y 29.372,Z 195.624,A -5.813,B 90.000,C 0.000} C_DIS
LIN {X -288.498,Y 29.473,Z 195.700,A -5.833,B 90.000,C 0.000} C_DIS
LIN {X -288.496,Y 29.495,Z 195.791,A -5.837,B 90.000,C 0.000} C_DIS
LIN {X -288.492,Y 29.537,Z 195.912,A -5.846,B 90.000,C 0.000} C_DIS
LIN {X -288.471,Y 29.740,Z 196.130,A -5.886,B 90.000,C 0.000} C_DIS
LIN {X -288.462,Y 29.824,Z 196.350,A -5.903,B 90.000,C 0.000} C_DIS
LIN {X -288.441,Y 30.027,Z 196.563,A -5.943,B 90.000,C 0.000} C_DIS
LIN {X -288.432,Y 30.112,Z 196.784,A -5.960,B 90.000,C 0.000} C_DIS
LIN {X -288.411,Y 30.315,Z 197.002,A -6.000,B 90.000,C 0.000} C_DIS
LIN {X -288.407,Y 30.357,Z 197.123,A -6.009,B 90.000,C 0.000} C_DIS
LIN {X -288.405,Y 30.378,Z 197.214,A -6.013,B 90.000,C 0.000} C_DIS
LIN {X -288.394,Y 30.480,Z 197.290,A -6.033,B 90.000,C 0.000} C_DIS
LIN {X -288.392,Y 30.501,Z 197.380,A -6.037,B 90.000,C 0.000} C_DIS
LIN {X -288.387,Y 30.543,Z 197.502,A -6.046,B 90.000,C 0.000} C_DIS
LIN {X -288.366,Y 30.746,Z 197.720,A -6.086,B 90.000,C 0.000} C_DIS
LIN {X -288.357,Y 30.830,Z 197.940,A -6.103,B 90.000,C 0.000} C_DIS
LIN {X -288.335,Y 31.033,Z 198.158,A -6.143,B 90.000,C 0.000} C_DIS
LIN {X -288.330,Y 31.076,Z 198.279,A -6.151,B 90.000,C 0.000} C_DIS
LIN {X -288.328,Y 31.097,Z 198.370,A -6.156,B 90.000,C 0.000} C_DIS
LIN {X -288.317,Y 31.198,Z 198.446,A -6.176,B 90.000,C 0.000} C_DIS
LIN {X -288.315,Y 31.219,Z 198.537,A -6.180,B 90.000,C 0.000} C_DIS
LIN {X -288.310,Y 31.262,Z 198.658,A -6.188,B 90.000,C 0.000} C_DIS
LIN {X -288.288,Y 31.464,Z 198.876,A -6.229,B 90.000,C 0.000} C_DIS
LIN {X -288.279,Y 31.549,Z 199.096,A -6.246,B 90.000,C 0.000} C_DIS
LIN {X -288.257,Y 31.752,Z 199.310,A -6.286,B 90.000,C 0.000} C_DIS
LIN {X -288.247,Y 31.836,Z 199.530,A -6.303,B 90.000,C 0.000} C_DIS
LIN {X -288.225,Y 32.039,Z 199.748,A -6.343,B 90.000,C 0.000} C_DIS
LIN {X -288.220,Y 32.081,Z 199.869,A -6.351,B 90.000,C 0.000} C_DIS
LIN {X -288.218,Y 32.102,Z 199.960,A -6.356,B 90.000,C 0.000} C_DIS
LIN {X -288.206,Y 32.204,Z 200.036,A -6.376,B 90.000,C 0.000} C_DIS
LIN {X -288.204,Y 32.225,Z 200.126,A -6.380,B 90.000,C 0.000} C_DIS
LIN {X -288.199,Y 32.267,Z 200.248,A -6.388,B 90.000,C 0.000} C_DIS
LIN {X -288.177,Y 32.470,Z 200.466,A -6.429,B 90.000,C 0.000} C_DIS
LIN {X -288.167,Y 32.554,Z 200.686,A -6.445,B 90.000,C 0.000} C_DIS
LIN {X -288.144,Y 32.757,Z 200.904,A -6.486,B 90.000,C 0.000} C_DIS
LIN {X -288.139,Y 32.799,Z 201.025,A -6.494,B 90.000,C 0.000} C_DIS
LIN {X -288.137,Y 32.821,Z 201.116,A -6.498,B 90.000,C 0.000} C_DIS
LIN {X -288.125,Y 32.922,Z 201.192,A -6.518,B 90.000,C 0.000} C_DIS
LIN {X -288.123,Y 32.943,Z 201.283,A -6.523,B 90.000,C 0.000} C_DIS
LIN {X -288.118,Y 32.985,Z 201.404,A -6.531,B 90.000,C 0.000} C_DIS
LIN {X -288.095,Y 33.188,Z 201.622,A -6.571,B 90.000,C 0.000} C_DIS
LIN {X -288.085,Y 33.272,Z 201.842,A -6.588,B 90.000,C 0.000} C_DIS
LIN {X -288.061,Y 33.475,Z 202.060,A -6.629,B 90.000,C 0.000} C_DIS
LIN {X -288.057,Y 33.517,Z 202.182,A -6.637,B 90.000,C 0.000} C_DIS
LIN {X -288.054,Y 33.538,Z 202.272,A -6.641,B 90.000,C 0.000} C_DIS
LIN {X -288.042,Y 33.640,Z 202.348,A -6.661,B 90.000,C 0.000} C_DIS
LIN {X -288.040,Y 33.661,Z 202.439,A -6.665,B 90.000,C 0.000} C_DIS
LIN {X -288.035,Y 33.703,Z 202.560,A -6.674,B 90.000,C 0.000} C_DIS
LIN {X -288.011,Y 33.906,Z 202.778,A -6.714,B 90.000,C 0.000} C_DIS
LIN {X -288.001,Y 33.990,Z 202.998,A -6.731,B 90.000,C 0.000} C_DIS
LIN {X -287.977,Y 34.193,Z 203.212,A -6.771,B 90.000,C 0.000} C_DIS
LIN {X -287.967,Y 34.277,Z 203.432,A -6.788,B 90.000,C 0.000} C_DIS
LIN {X -287.943,Y 34.480,Z 203.650,A -6.828,B 90.000,C 0.000} C_DIS
LIN {X -287.938,Y 34.522,Z 203.771,A -6.837,B 90.000,C 0.000} C_DIS
LIN {X -287.935,Y 34.543,Z 203.862,A -6.841,B 90.000,C 0.000} C_DIS
LIN {X -287.923,Y 34.644,Z 203.938,A -6.861,B 90.000,C 0.000} C_DIS
LIN {X -287.921,Y 34.666,Z 204.029,A -6.865,B 90.000,C 0.000} C_DIS
LIN {X -287.916,Y 34.708,Z 204.150,A -6.874,B 90.000,C 0.000} C_DIS
LIN {X -287.891,Y 34.910,Z 204.368,A -6.914,B 90.000,C 0.000} C_DIS
LIN {X -287.881,Y 34.995,Z 204.588,A -6.931,B 90.000,C 0.000} C_DIS
LIN {X -287.856,Y 35.197,Z 204.806,A -6.971,B 90.000,C 0.000} C_DIS
LIN {X -287.851,Y 35.239,Z 204.928,A -6.980,B 90.000,C 0.000} C_DIS
LIN {X -287.848,Y 35.260,Z 205.018,A -6.984,B 90.000,C 0.000} C_DIS
LIN {X -287.836,Y 35.362,Z 205.094,A -7.004,B 90.000,C 0.000} C_DIS
LIN {X -287.833,Y 35.383,Z 205.185,A -7.008,B 90.000,C 0.000} C_DIS
LIN {X -287.828,Y 35.425,Z 205.306,A -7.017,B 90.000,C 0.000} C_DIS
LIN {X -287.803,Y 35.628,Z 205.524,A -7.057,B 90.000,C 0.000} C_DIS
LIN {X -287.793,Y 35.712,Z 205.745,A -7.074,B 90.000,C 0.000} C_DIS
LIN {X -287.768,Y 35.914,Z 205.958,A -7.114,B 90.000,C 0.000} C_DIS
LIN {X -287.757,Y 35.999,Z 206.178,A -7.131,B 90.000,C 0.000} C_DIS
LIN {X -287.732,Y 36.201,Z 206.396,A -7.171,B 90.000,C 0.000} C_DIS
LIN {X -287.726,Y 36.243,Z 206.517,A -7.179,B 90.000,C 0.000} C_DIS
LIN {X -287.724,Y 36.264,Z 206.608,A -7.184,B 90.000,C 0.000} C_DIS
LIN {X -287.711,Y 36.366,Z 206.684,A -7.204,B 90.000,C 0.000} C_DIS
LIN {X -287.708,Y 36.387,Z 206.775,A -7.208,B 90.000,C 0.000} C_DIS
LIN {X -287.703,Y 36.429,Z 206.896,A -7.216,B 90.000,C 0.000} C_DIS
LIN {X -287.677,Y 36.631,Z 207.114,A -7.257,B 90.000,C 0.000} C_DIS
LIN {X -287.666,Y 36.716,Z 207.334,A -7.273,B 90.000,C 0.000} C_DIS
LIN {X -287.640,Y 36.918,Z 207.552,A -7.314,B 90.000,C 0.000} C_DIS
LIN {X -287.635,Y 36.960,Z 207.674,A -7.322,B 90.000,C 0.000} C_DIS
LIN {X -287.632,Y 36.981,Z 207.765,A -7.326,B 90.000,C 0.000} C_DIS
LIN {X -287.619,Y 37.083,Z 207.840,A -7.347,B 90.000,C 0.000} C_DIS
LIN {X -287.617,Y 37.104,Z 207.931,A -7.351,B 90.000,C 0.000} C_DIS
LIN {X -287.611,Y 37.146,Z 208.052,A -7.359,B 90.000,C 0.000} C_DIS
LIN {X -287.585,Y 37.348,Z 208.270,A -7.399,B 90.000,C 0.000} C_DIS
LIN {X -287.574,Y 37.432,Z 208.491,A -7.416,B 90.000,C 0.000} C_DIS
LIN {X -287.548,Y 37.635,Z 208.709,A -7.457,B 90.000,C 0.000} C_DIS
LIN {X -287.542,Y 37.677,Z 208.830,A -7.465,B 90.000,C 0.000} C_DIS
LIN {X -287.539,Y 37.698,Z 208.921,A -7.469,B 90.000,C 0.000} C_DIS
LIN {X -287.526,Y 37.799,Z 208.996,A -7.489,B 90.000,C 0.000} C_DIS
LIN {X -287.523,Y 37.820,Z 209.087,A -7.494,B 90.000,C 0.000} C_DIS
LIN {X -287.518,Y 37.862,Z 209.209,A -7.502,B 90.000,C 0.000} C_DIS
LIN {X -287.491,Y 38.065,Z 209.426,A -7.542,B 90.000,C 0.000} C_DIS
LIN {X -287.480,Y 38.149,Z 209.647,A -7.559,B 90.000,C 0.000} C_DIS
LIN {X -287.453,Y 38.351,Z 209.860,A -7.599,B 90.000,C 0.000} C_DIS
LIN {X -287.442,Y 38.435,Z 210.080,A -7.616,B 90.000,C 0.000} C_DIS
LIN {X -287.415,Y 38.638,Z 210.298,A -7.656,B 90.000,C 0.000} C_DIS
LIN {X -287.409,Y 38.680,Z 210.420,A -7.665,B 90.000,C 0.000} C_DIS
LIN {X -287.406,Y 38.701,Z 210.511,A -7.669,B 90.000,C 0.000} C_DIS
LIN {X -287.392,Y 38.802,Z 210.586,A -7.689,B 90.000,C 0.000} C_DIS
LIN {X -287.390,Y 38.823,Z 210.677,A -7.693,B 90.000,C 0.000} C_DIS
LIN {X -287.384,Y 38.865,Z 210.798,A -7.702,B 90.000,C 0.000} C_DIS
LIN {X -287.356,Y 39.067,Z 211.016,A -7.742,B 90.000,C 0.000} C_DIS
LIN {X -287.345,Y 39.152,Z 211.237,A -7.759,B 90.000,C 0.000} C_DIS
LIN {X -287.317,Y 39.354,Z 211.455,A -7.799,B 90.000,C 0.000} C_DIS
LIN {X -287.312,Y 39.396,Z 211.576,A -7.808,B 90.000,C 0.000} C_DIS
LIN {X -287.309,Y 39.417,Z 211.667,A -7.812,B 90.000,C 0.000} C_DIS
LIN {X -287.295,Y 39.518,Z 211.742,A -7.832,B 90.000,C 0.000} C_DIS
LIN {X -287.292,Y 39.539,Z 211.833,A -7.836,B 90.000,C 0.000} C_DIS
LIN {X -287.286,Y 39.581,Z 211.955,A -7.845,B 90.000,C 0.000} C_DIS
LIN {X -287.258,Y 39.783,Z 212.173,A -7.885,B 90.000,C 0.000} C_DIS
LIN {X -287.247,Y 39.867,Z 212.393,A -7.902,B 90.000,C 0.000} C_DIS
LIN {X -287.218,Y 40.070,Z 212.606,A -7.942,B 90.000,C 0.000} C_DIS
LIN {X -287.207,Y 40.154,Z 212.826,A -7.959,B 90.000,C 0.000} C_DIS
LIN {X -287.178,Y 40.356,Z 213.044,A -7.999,B 90.000,C 0.000} C_DIS
LIN {X -287.172,Y 40.398,Z 213.166,A -8.008,B 90.000,C 0.000} C_DIS
LIN {X -287.169,Y 40.419,Z 213.257,A -8.012,B 90.000,C 0.000} C_DIS
LIN {X -287.155,Y 40.520,Z 213.332,A -8.032,B 90.000,C 0.000} C_DIS
LIN {X -287.152,Y 40.541,Z 213.423,A -8.036,B 90.000,C 0.000} C_DIS
LIN {X -287.146,Y 40.583,Z 213.544,A -8.044,B 90.000,C 0.000} C_DIS
LIN {X -287.118,Y 40.785,Z 213.762,A -8.085,B 90.000,C 0.000} C_DIS
LIN {X -287.106,Y 40.869,Z 213.983,A -8.102,B 90.000,C 0.000} C_DIS
LIN {X -287.077,Y 41.071,Z 214.196,A -8.142,B 90.000,C 0.000} C_DIS
LIN {X -287.065,Y 41.155,Z 214.416,A -8.159,B 90.000,C 0.000} C_DIS
LIN {X -287.036,Y 41.358,Z 214.634,A -8.199,B 90.000,C 0.000} C_DIS
LIN {X -287.030,Y 41.400,Z 214.756,A -8.207,B 90.000,C 0.000} C_DIS
LIN {X -287.027,Y 41.421,Z 214.846,A -8.212,B 90.000,C 0.000} C_DIS
LIN {X -287.012,Y 41.522,Z 214.922,A -8.232,B 90.000,C 0.000} C_DIS
LIN {X -287.009,Y 41.543,Z 215.013,A -8.236,B 90.000,C 0.000} C_DIS
LIN {X -287.003,Y 41.585,Z 215.134,A -8.244,B 90.000,C 0.000} C_DIS
LIN {X -286.974,Y 41.787,Z 215.352,A -8.285,B 90.000,C 0.000} C_DIS
LIN {X -286.961,Y 41.871,Z 215.572,A -8.301,B 90.000,C 0.000} C_DIS
LIN {X -286.932,Y 42.073,Z 215.790,A -8.342,B 90.000,C 0.000} C_DIS
LIN {X -286.926,Y 42.115,Z 215.912,A -8.350,B 90.000,C 0.000} C_DIS
LIN {X -286.923,Y 42.136,Z 216.003,A -8.354,B 90.000,C 0.000} C_DIS
LIN {X -286.908,Y 42.237,Z 216.078,A -8.375,B 90.000,C 0.000} C_DIS
LIN {X -286.905,Y 42.258,Z 216.169,A -8.379,B 90.000,C 0.000} C_DIS
LIN {X -286.898,Y 42.300,Z 216.290,A -8.387,B 90.000,C 0.000} C_DIS
LIN {X -286.869,Y 42.502,Z 216.508,A -8.427,B 90.000,C 0.000} C_DIS
LIN {X -286.856,Y 42.586,Z 216.729,A -8.444,B 90.000,C 0.000} C_DIS
LIN {X -286.826,Y 42.787,Z 216.947,A -8.485,B 90.000,C 0.000} C_DIS
LIN {X -286.820,Y 42.829,Z 217.068,A -8.493,B 90.000,C 0.000} C_DIS
LIN {X -286.817,Y 42.850,Z 217.159,A -8.497,B 90.000,C 0.000} C_DIS
LIN {X -286.802,Y 42.951,Z 217.234,A -8.517,B 90.000,C 0.000} C_DIS
LIN {X -286.798,Y 42.972,Z 217.325,A -8.522,B 90.000,C 0.000} C_DIS
LIN {X -286.792,Y 43.014,Z 217.447,A -8.530,B 90.000,C 0.000} C_DIS
LIN {X -286.762,Y 43.216,Z 217.665,A -8.570,B 90.000,C 0.000} C_DIS
LIN {X -286.749,Y 43.300,Z 217.885,A -8.587,B 90.000,C 0.000} C_DIS
LIN {X -286.719,Y 43.502,Z 218.098,A -8.627,B 90.000,C 0.000} C_DIS
LIN {X -286.706,Y 43.586,Z 218.318,A -8.644,B 90.000,C 0.000} C_DIS
LIN {X -286.675,Y 43.788,Z 218.536,A -8.684,B 90.000,C 0.000} C_DIS
LIN {X -286.669,Y 43.830,Z 218.658,A -8.693,B 90.000,C 0.000} C_DIS
LIN {X -286.665,Y 43.851,Z 218.749,A -8.697,B 90.000,C 0.000} C_DIS
LIN {X -286.650,Y 43.952,Z 218.824,A -8.717,B 90.000,C 0.000} C_DIS
LIN {X -286.647,Y 43.973,Z 218.915,A -8.721,B 90.000,C 0.000} C_DIS
LIN {X -286.640,Y 44.015,Z 219.036,A -8.730,B 90.000,C 0.000} C_DIS
LIN {X -286.609,Y 44.216,Z 219.254,A -8.770,B 90.000,C 0.000} C_DIS
LIN {X -286.596,Y 44.300,Z 219.475,A -8.787,B 90.000,C 0.000} C_DIS
LIN {X -286.565,Y 44.502,Z 219.693,A -8.827,B 90.000,C 0.000} C_DIS
LIN {X -286.559,Y 44.544,Z 219.814,A -8.836,B 90.000,C 0.000} C_DIS
LIN {X -286.555,Y 44.565,Z 219.905,A -8.840,B 90.000,C 0.000} C_DIS
LIN {X -286.540,Y 44.666,Z 219.980,A -8.860,B 90.000,C 0.000} C_DIS
LIN {X -286.536,Y 44.687,Z 220.071,A -8.864,B 90.000,C 0.000} C_DIS
LIN {X -286.530,Y 44.729,Z 220.193,A -8.873,B 90.000,C 0.000} C_DIS
LIN {X -286.498,Y 44.930,Z 220.411,A -8.913,B 90.000,C 0.000} C_DIS
LIN {X -286.485,Y 45.014,Z 220.631,A -8.930,B 90.000,C 0.000} C_DIS
LIN {X -286.453,Y 45.216,Z 220.849,A -8.970,B 90.000,C 0.000} C_DIS
LIN {X -286.447,Y 45.258,Z 220.970,A -8.978,B 90.000,C 0.000} C_DIS
LIN {X -286.443,Y 45.279,Z 221.061,A -8.983,B 90.000,C 0.000} C_DIS
LIN {X -286.427,Y 45.380,Z 221.137,A -9.003,B 90.000,C 0.000} C_DIS
LIN {X -286.424,Y 45.401,Z 221.227,A -9.007,B 90.000,C 0.000} C_DIS
LIN {X -286.417,Y 45.443,Z 221.349,A -9.015,B 90.000,C 0.000} C_DIS
LIN {X -286.385,Y 45.644,Z 221.567,A -9.056,B 90.000,C 0.000} C_DIS
LIN {X -286.372,Y 45.728,Z 221.787,A -9.072,B 90.000,C 0.000} C_DIS
LIN {X -286.340,Y 45.930,Z 222.000,A -9.113,B 90.000,C 0.000} C_DIS
LIN {X -286.326,Y 46.014,Z 222.221,A -9.130,B 90.000,C 0.000} C_DIS
LIN {X -286.294,Y 46.215,Z 222.439,A -9.170,B 90.000,C 0.000} C_DIS
LIN {X -286.287,Y 46.257,Z 222.560,A -9.178,B 90.000,C 0.000} C_DIS
LIN {X -286.284,Y 46.278,Z 222.651,A -9.182,B 90.000,C 0.000} C_DIS
LIN {X -286.267,Y 46.379,Z 222.731,A -9.203,B 90.000,C 0.000} C_DIS
LIN {X -286.261,Y 46.421,Z 222.935,A -9.211,B 90.000,C 0.000} C_DIS
LIN {X -286.244,Y 46.521,Z 223.020,A -9.231,B 90.000,C 0.000} C_DIS
LIN {X -286.237,Y 46.563,Z 223.224,A -9.240,B 90.000,C 0.000} C_DIS
LIN {X -286.229,Y 46.614,Z 223.267,A -9.250,B 90.000,C 0.000} C_DIS
LIN {X -286.221,Y 46.664,Z 223.373,A -9.260,B 90.000,C 0.000} C_DIS
LIN {X -286.214,Y 46.706,Z 223.883,A -9.268,B 90.000,C 0.000} C_DIS
LIN {X -286.198,Y 46.807,Z 224.086,A -9.288,B 90.000,C 0.000} C_DIS
LIN {X -286.188,Y 46.869,Z 224.587,A -9.301,B 90.000,C 0.000} C_DIS
LIN {X -286.169,Y 46.981,Z 224.803,A -9.323,B 90.000,C 0.000} C_DIS
LIN {X -286.141,Y 47.150,Z 224.948,A -9.357,B 90.000,C 0.000} C_DIS
LIN {X -286.086,Y 47.487,Z 225.022,A -9.425,B 90.000,C 0.000} C_DIS
LIN {X -286.077,Y 47.541,Z 225.073,A -9.435,B 90.000,C 0.000} C_DIS
LIN {X -286.071,Y 47.573,Z 225.124,A -9.442,B 90.000,C 0.000} C_DIS
LIN {X -286.058,Y 47.651,Z 225.146,A -9.457,B 90.000,C 0.000} C_DIS
LIN {X -286.037,Y 47.779,Z 225.198,A -9.483,B 90.000,C 0.000} C_DIS
LIN {X -286.012,Y 47.931,Z 225.321,A -9.514,B 90.000,C 0.000} C_DIS
LIN {X -285.990,Y 48.058,Z 225.470,A -9.539,B 90.000,C 0.000} C_DIS
LIN {X -285.981,Y 48.111,Z 225.596,A -9.549,B 90.000,C 0.000} C_DIS
LIN {X -285.957,Y 48.253,Z 225.796,A -9.578,B 90.000,C 0.000} C_DIS
LIN {X -285.940,Y 48.354,Z 225.903,A -9.598,B 90.000,C 0.000} C_DIS
LIN {X -285.926,Y 48.438,Z 226.123,A -9.615,B 90.000,C 0.000} C_DIS
LIN {X -285.892,Y 48.639,Z 226.341,A -9.655,B 90.000,C 0.000} C_DIS
LIN {X -285.885,Y 48.681,Z 226.462,A -9.664,B 90.000,C 0.000} C_DIS
LIN {X -285.881,Y 48.702,Z 226.553,A -9.668,B 90.000,C 0.000} C_DIS
LIN {X -285.864,Y 48.802,Z 226.629,A -9.688,B 90.000,C 0.000} C_DIS
LIN {X -285.861,Y 48.823,Z 226.720,A -9.692,B 90.000,C 0.000} C_DIS
LIN {X -285.853,Y 48.865,Z 226.841,A -9.701,B 90.000,C 0.000} C_DIS
LIN {X -285.819,Y 49.066,Z 227.059,A -9.741,B 90.000,C 0.000} C_DIS
LIN {X -285.805,Y 49.150,Z 227.279,A -9.758,B 90.000,C 0.000} C_DIS
LIN {X -285.770,Y 49.351,Z 227.493,A -9.798,B 90.000,C 0.000} C_DIS
LIN {X -285.755,Y 49.435,Z 227.713,A -9.815,B 90.000,C 0.000} C_DIS
LIN {X -285.721,Y 49.636,Z 227.931,A -9.855,B 90.000,C 0.000} C_DIS
LIN {X -285.713,Y 49.678,Z 228.052,A -9.864,B 90.000,C 0.000} C_DIS
LIN {X -285.710,Y 49.699,Z 228.143,A -9.868,B 90.000,C 0.000} C_DIS
LIN {X -285.692,Y 49.799,Z 228.219,A -9.888,B 90.000,C 0.000} C_DIS
LIN {X -285.689,Y 49.820,Z 228.309,A -9.892,B 90.000,C 0.000} C_DIS
LIN {X -285.681,Y 49.862,Z 228.431,A -9.901,B 90.000,C 0.000} C_DIS
LIN {X -285.646,Y 50.063,Z 228.649,A -9.941,B 90.000,C 0.000} C_DIS
LIN {X -285.631,Y 50.147,Z 228.869,A -9.958,B 90.000,C 0.000} C_DIS
LIN {X -285.596,Y 50.348,Z 229.087,A -9.998,B 90.000,C 0.000} C_DIS
LIN {X -285.589,Y 50.390,Z 229.208,A -10.006,B 90.000,C 0.000} C_DIS
LIN {X -285.585,Y 50.411,Z 229.299,A -10.011,B 90.000,C 0.000} C_DIS
LIN {X -285.567,Y 50.511,Z 229.375,A -10.031,B 90.000,C 0.000} C_DIS
LIN {X -285.564,Y 50.532,Z 229.466,A -10.035,B 90.000,C 0.000} C_DIS
LIN {X -285.556,Y 50.574,Z 229.587,A -10.043,B 90.000,C 0.000} C_DIS
LIN {X -285.520,Y 50.775,Z 229.805,A -10.084,B 90.000,C 0.000} C_DIS
LIN {X -285.506,Y 50.858,Z 230.025,A -10.100,B 90.000,C 0.000} C_DIS
LIN {X -285.470,Y 51.059,Z 230.243,A -10.141,B 90.000,C 0.000} C_DIS
LIN {X -285.462,Y 51.101,Z 230.365,A -10.149,B 90.000,C 0.000} C_DIS
LIN {X -285.458,Y 51.122,Z 230.455,A -10.153,B 90.000,C 0.000} C_DIS
LIN {X -285.440,Y 51.223,Z 230.531,A -10.173,B 90.000,C 0.000} C_DIS
LIN {X -285.437,Y 51.243,Z 230.622,A -10.178,B 90.000,C 0.000} C_DIS
LIN {X -285.429,Y 51.285,Z 230.743,A -10.186,B 90.000,C 0.000} C_DIS
LIN {X -285.393,Y 51.486,Z 230.961,A -10.226,B 90.000,C 0.000} C_DIS
LIN {X -285.378,Y 51.570,Z 231.181,A -10.243,B 90.000,C 0.000} C_DIS
LIN {X -285.342,Y 51.771,Z 231.395,A -10.284,B 90.000,C 0.000} C_DIS
LIN {X -285.326,Y 51.854,Z 231.615,A -10.300,B 90.000,C 0.000} C_DIS
LIN {X -285.290,Y 52.055,Z 231.833,A -10.341,B 90.000,C 0.000} C_DIS
LIN {X -285.282,Y 52.097,Z 231.954,A -10.349,B 90.000,C 0.000} C_DIS
LIN {X -285.278,Y 52.118,Z 232.045,A -10.353,B 90.000,C 0.000} C_DIS
LIN {X -285.260,Y 52.218,Z 232.121,A -10.373,B 90.000,C 0.000} C_DIS
LIN {X -285.256,Y 52.239,Z 232.212,A -10.378,B 90.000,C 0.000} C_DIS
LIN {X -285.249,Y 52.281,Z 232.333,A -10.386,B 90.000,C 0.000} C_DIS
LIN {X -285.212,Y 52.481,Z 232.551,A -10.426,B 90.000,C 0.000} C_DIS
LIN {X -285.196,Y 52.565,Z 232.771,A -10.443,B 90.000,C 0.000} C_DIS
LIN {X -285.159,Y 52.766,Z 232.989,A -10.483,B 90.000,C 0.000} C_DIS
LIN {X -285.151,Y 52.807,Z 233.111,A -10.492,B 90.000,C 0.000} C_DIS
LIN {X -285.148,Y 52.828,Z 233.201,A -10.496,B 90.000,C 0.000} C_DIS
LIN {X -285.129,Y 52.929,Z 233.277,A -10.516,B 90.000,C 0.000} C_DIS
LIN {X -285.125,Y 52.950,Z 233.368,A -10.520,B 90.000,C 0.000} C_DIS
LIN {X -285.117,Y 52.991,Z 233.489,A -10.529,B 90.000,C 0.000} C_DIS
LIN {X -285.080,Y 53.192,Z 233.707,A -10.569,B 90.000,C 0.000} C_DIS
LIN {X -285.064,Y 53.275,Z 233.928,A -10.586,B 90.000,C 0.000} C_DIS
LIN {X -285.027,Y 53.476,Z 234.141,A -10.626,B 90.000,C 0.000} C_DIS
LIN {X -285.011,Y 53.560,Z 234.361,A -10.643,B 90.000,C 0.000} C_DIS
LIN {X -284.973,Y 53.760,Z 234.579,A -10.683,B 90.000,C 0.000} C_DIS
LIN {X -284.966,Y 53.802,Z 234.700,A -10.692,B 90.000,C 0.000} C_DIS
LIN {X -284.962,Y 53.823,Z 234.791,A -10.696,B 90.000,C 0.000} C_DIS
LIN {X -284.943,Y 53.923,Z 234.867,A -10.716,B 90.000,C 0.000} C_DIS
LIN {X -284.939,Y 53.944,Z 234.958,A -10.720,B 90.000,C 0.000} C_DIS
LIN {X -284.931,Y 53.986,Z 235.079,A -10.729,B 90.000,C 0.000} C_DIS
LIN {X -284.893,Y 54.186,Z 235.297,A -10.769,B 90.000,C 0.000} C_DIS
LIN {X -284.877,Y 54.270,Z 235.517,A -10.786,B 90.000,C 0.000} C_DIS
LIN {X -284.839,Y 54.470,Z 235.735,A -10.826,B 90.000,C 0.000} C_DIS
LIN {X -284.831,Y 54.512,Z 235.857,A -10.834,B 90.000,C 0.000} C_DIS
LIN {X -284.827,Y 54.533,Z 235.948,A -10.839,B 90.000,C 0.000} C_DIS
LIN {X -284.807,Y 54.633,Z 236.019,A -10.859,B 90.000,C 0.000} C_DIS
LIN {X -284.798,Y 54.683,Z 236.210,A -10.869,B 90.000,C 0.000} C_DIS
LIN {X -284.784,Y 54.757,Z 236.314,A -10.884,B 90.000,C 0.000} C_DIS
LIN {X -284.764,Y 54.858,Z 236.389,A -10.904,B 90.000,C 0.000} C_DIS
LIN {X -284.728,Y 55.047,Z 236.440,A -10.942,B 90.000,C 0.000} C_DIS
LIN {X -284.721,Y 55.080,Z 236.491,A -10.949,B 90.000,C 0.000} C_DIS
LIN {X -284.705,Y 55.163,Z 236.542,A -10.965,B 90.000,C 0.000} C_DIS
LIN {X -284.666,Y 55.363,Z 236.563,A -11.006,B 90.000,C 0.000} C_DIS
LIN {X -284.627,Y 55.564,Z 236.542,A -11.046,B 90.000,C 0.000} C_DIS
LIN {X -284.611,Y 55.647,Z 236.491,A -11.063,B 90.000,C 0.000} C_DIS
LIN {X -284.603,Y 55.689,Z 236.440,A -11.071,B 90.000,C 0.000} C_DIS
LIN {X -284.583,Y 55.789,Z 236.419,A -11.091,B 90.000,C 0.000} C_DIS
LIN {X -284.562,Y 55.895,Z 236.383,A -11.113,B 90.000,C 0.000} C_DIS
LIN {X -284.555,Y 55.931,Z 236.274,A -11.120,B 90.000,C 0.000} C_DIS
LIN {X -284.551,Y 55.951,Z 236.172,A -11.124,B 90.000,C 0.000} C_DIS
LIN {X -284.541,Y 56.002,Z 236.130,A -11.134,B 90.000,C 0.000} C_DIS
LIN {X -284.532,Y 56.052,Z 236.045,A -11.144,B 90.000,C 0.000} C_DIS
LIN {X -284.523,Y 56.093,Z 235.637,A -11.153,B 90.000,C 0.000} C_DIS
LIN {X -284.513,Y 56.143,Z 235.552,A -11.163,B 90.000,C 0.000} C_DIS
LIN {X -284.503,Y 56.194,Z 235.407,A -11.173,B 90.000,C 0.000} C_DIS
LIN {X -284.495,Y 56.235,Z 234.685,A -11.181,B 90.000,C 0.000} C_DIS
LIN {X -284.475,Y 56.336,Z 234.395,A -11.202,B 90.000,C 0.000} C_DIS
LIN {X -284.467,Y 56.376,Z 233.673,A -11.210,B 90.000,C 0.000} C_DIS
LIN {X -284.447,Y 56.478,Z 233.384,A -11.230,B 90.000,C 0.000} C_DIS
LIN {X -284.439,Y 56.518,Z 232.661,A -11.238,B 90.000,C 0.000} C_DIS
LIN {X -284.419,Y 56.619,Z 232.390,A -11.259,B 90.000,C 0.000} C_DIS
LIN {X -284.411,Y 56.660,Z 231.776,A -11.267,B 90.000,C 0.000} C_DIS
LIN {X -284.391,Y 56.761,Z 231.505,A -11.287,B 90.000,C 0.000} C_DIS
LIN {X -284.383,Y 56.802,Z 230.782,A -11.295,B 90.000,C 0.000} C_DIS
LIN {X -284.363,Y 56.902,Z 230.511,A -11.316,B 90.000,C 0.000} C_DIS
LIN {X -284.354,Y 56.944,Z 229.897,A -11.324,B 90.000,C 0.000} C_DIS
LIN {X -284.334,Y 57.044,Z 229.626,A -11.344,B 90.000,C 0.000} C_DIS
LIN {X -284.326,Y 57.085,Z 228.903,A -11.353,B 90.000,C 0.000} C_DIS
LIN {X -284.306,Y 57.186,Z 228.614,A -11.373,B 90.000,C 0.000} C_DIS
LIN {X -284.298,Y 57.227,Z 227.892,A -11.381,B 90.000,C 0.000} C_DIS
LIN {X -284.277,Y 57.328,Z 227.603,A -11.401,B 90.000,C 0.000} C_DIS
LIN {X -284.269,Y 57.368,Z 226.880,A -11.410,B 90.000,C 0.000} C_DIS
LIN {X -284.249,Y 57.469,Z 226.609,A -11.430,B 90.000,C 0.000} C_DIS
LIN {X -284.240,Y 57.510,Z 225.995,A -11.438,B 90.000,C 0.000} C_DIS
LIN {X -284.220,Y 57.611,Z 225.724,A -11.459,B 90.000,C 0.000} C_DIS
LIN {X -284.212,Y 57.652,Z 225.001,A -11.467,B 90.000,C 0.000} C_DIS
LIN {X -284.191,Y 57.752,Z 224.730,A -11.487,B 90.000,C 0.000} C_DIS
LIN {X -284.183,Y 57.794,Z 224.116,A -11.495,B 90.000,C 0.000} C_DIS
LIN {X -284.162,Y 57.894,Z 223.845,A -11.516,B 90.000,C 0.000} C_DIS
LIN {X -284.154,Y 57.935,Z 223.122,A -11.524,B 90.000,C 0.000} C_DIS
LIN {X -284.133,Y 58.036,Z 222.833,A -11.544,B 90.000,C 0.000} C_DIS
LIN {X -284.125,Y 58.077,Z 222.111,A -11.552,B 90.000,C 0.000} C_DIS
LIN {X -284.105,Y 58.177,Z 221.840,A -11.573,B 90.000,C 0.000} C_DIS
LIN {X -284.096,Y 58.219,Z 221.225,A -11.581,B 90.000,C 0.000} C_DIS
LIN {X -284.075,Y 58.319,Z 220.954,A -11.601,B 90.000,C 0.000} C_DIS
LIN {X -284.067,Y 58.360,Z 220.232,A -11.610,B 90.000,C 0.000} C_DIS
LIN {X -284.046,Y 58.461,Z 219.943,A -11.630,B 90.000,C 0.000} C_DIS
LIN {X -284.038,Y 58.501,Z 219.220,A -11.638,B 90.000,C 0.000} C_DIS
LIN {X -284.017,Y 58.602,Z 218.949,A -11.658,B 90.000,C 0.000} C_DIS
LIN {X -284.009,Y 58.643,Z 218.335,A -11.667,B 90.000,C 0.000} C_DIS
LIN {X -283.988,Y 58.744,Z 218.064,A -11.687,B 90.000,C 0.000} C_DIS
LIN {X -283.980,Y 58.784,Z 217.341,A -11.695,B 90.000,C 0.000} C_DIS
LIN {X -283.959,Y 58.885,Z 217.070,A -11.715,B 90.000,C 0.000} C_DIS
LIN {X -283.950,Y 58.926,Z 216.456,A -11.724,B 90.000,C 0.000} C_DIS
LIN {X -283.929,Y 59.027,Z 216.185,A -11.744,B 90.000,C 0.000} C_DIS
LIN {X -283.921,Y 59.067,Z 215.462,A -11.752,B 90.000,C 0.000} C_DIS
LIN {X -283.900,Y 59.168,Z 215.173,A -11.773,B 90.000,C 0.000} C_DIS
LIN {X -283.891,Y 59.209,Z 214.451,A -11.781,B 90.000,C 0.000} C_DIS
LIN {X -283.870,Y 59.310,Z 214.162,A -11.801,B 90.000,C 0.000} C_DIS
LIN {X -283.862,Y 59.350,Z 213.439,A -11.809,B 90.000,C 0.000} C_DIS
LIN {X -283.841,Y 59.451,Z 213.168,A -11.830,B 90.000,C 0.000} C_DIS
LIN {X -283.832,Y 59.492,Z 212.554,A -11.838,B 90.000,C 0.000} C_DIS
LIN {X -283.811,Y 59.593,Z 212.283,A -11.858,B 90.000,C 0.000} C_DIS
LIN {X -283.803,Y 59.633,Z 211.560,A -11.866,B 90.000,C 0.000} C_DIS
LIN {X -283.781,Y 59.734,Z 211.289,A -11.887,B 90.000,C 0.000} C_DIS
LIN {X -283.773,Y 59.775,Z 210.675,A -11.895,B 90.000,C 0.000} C_DIS
LIN {X -283.751,Y 59.876,Z 210.404,A -11.915,B 90.000,C 0.000} C_DIS
LIN {X -283.743,Y 59.916,Z 209.681,A -11.924,B 90.000,C 0.000} C_DIS
LIN {X -283.722,Y 60.017,Z 209.392,A -11.944,B 90.000,C 0.000} C_DIS
LIN {X -283.713,Y 60.058,Z 208.669,A -11.952,B 90.000,C 0.000} C_DIS
LIN {X -283.692,Y 60.159,Z 208.380,A -11.973,B 90.000,C 0.000} C_DIS
LIN {X -283.683,Y 60.199,Z 207.658,A -11.981,B 90.000,C 0.000} C_DIS
LIN {X -283.662,Y 60.299,Z 207.387,A -12.001,B 90.000,C 0.000} C_DIS
LIN {X -283.653,Y 60.341,Z 206.773,A -12.009,B 90.000,C 0.000} C_DIS
LIN {X -283.632,Y 60.441,Z 206.502,A -12.030,B 90.000,C 0.000} C_DIS
LIN {X -283.623,Y 60.482,Z 205.779,A -12.038,B 90.000,C 0.000} C_DIS
LIN {X -283.601,Y 60.582,Z 205.508,A -12.058,B 90.000,C 0.000} C_DIS
LIN {X -283.593,Y 60.623,Z 204.894,A -12.066,B 90.000,C 0.000} C_DIS
LIN {X -283.571,Y 60.724,Z 204.623,A -12.087,B 90.000,C 0.000} C_DIS
LIN {X -283.563,Y 60.764,Z 203.900,A -12.095,B 90.000,C 0.000} C_DIS
LIN {X -283.541,Y 60.865,Z 203.611,A -12.115,B 90.000,C 0.000} C_DIS
LIN {X -283.532,Y 60.906,Z 202.888,A -12.123,B 90.000,C 0.000} C_DIS
LIN {X -283.511,Y 61.006,Z 202.617,A -12.144,B 90.000,C 0.000} C_DIS
LIN {X -283.502,Y 61.047,Z 202.003,A -12.152,B 90.000,C 0.000} C_DIS
LIN {X -283.480,Y 61.148,Z 201.732,A -12.172,B 90.000,C 0.000} C_DIS
LIN {X -283.471,Y 61.188,Z 201.009,A -12.181,B 90.000,C 0.000} C_DIS
LIN {X -283.450,Y 61.289,Z 200.720,A -12.201,B 90.000,C 0.000} C_DIS
LIN {X -283.441,Y 61.329,Z 199.998,A -12.209,B 90.000,C 0.000} C_DIS
LIN {X -283.419,Y 61.430,Z 199.727,A -12.229,B 90.000,C 0.000} C_DIS
LIN {X -283.410,Y 61.471,Z 199.113,A -12.238,B 90.000,C 0.000} C_DIS
LIN {X -283.388,Y 61.572,Z 198.842,A -12.258,B 90.000,C 0.000} C_DIS
LIN {X -283.380,Y 61.612,Z 198.119,A -12.266,B 90.000,C 0.000} C_DIS
LIN {X -283.358,Y 61.713,Z 197.830,A -12.287,B 90.000,C 0.000} C_DIS
LIN {X -283.349,Y 61.753,Z 197.107,A -12.295,B 90.000,C 0.000} C_DIS
LIN {X -283.327,Y 61.854,Z 196.836,A -12.315,B 90.000,C 0.000} C_DIS
LIN {X -283.318,Y 61.895,Z 196.222,A -12.323,B 90.000,C 0.000} C_DIS
LIN {X -283.296,Y 61.995,Z 195.951,A -12.344,B 90.000,C 0.000} C_DIS
LIN {X -283.287,Y 62.036,Z 195.228,A -12.352,B 90.000,C 0.000} C_DIS
LIN {X -283.265,Y 62.136,Z 194.957,A -12.372,B 90.000,C 0.000} C_DIS
LIN {X -283.256,Y 62.177,Z 194.343,A -12.381,B 90.000,C 0.000} C_DIS
LIN {X -283.234,Y 62.278,Z 194.072,A -12.401,B 90.000,C 0.000} C_DIS
LIN {X -283.225,Y 62.318,Z 193.349,A -12.409,B 90.000,C 0.000} C_DIS
LIN {X -283.203,Y 62.419,Z 193.060,A -12.429,B 90.000,C 0.000} C_DIS
LIN {X -283.194,Y 62.459,Z 192.338,A -12.438,B 90.000,C 0.000} C_DIS
LIN {X -283.172,Y 62.560,Z 192.049,A -12.458,B 90.000,C 0.000} C_DIS
LIN {X -283.163,Y 62.600,Z 191.326,A -12.466,B 90.000,C 0.000} C_DIS
LIN {X -283.141,Y 62.701,Z 191.055,A -12.486,B 90.000,C 0.000} C_DIS
LIN {X -283.132,Y 62.742,Z 190.441,A -12.495,B 90.000,C 0.000} C_DIS
LIN {X -283.109,Y 62.842,Z 190.170,A -12.515,B 90.000,C 0.000} C_DIS
LIN {X -283.100,Y 62.882,Z 189.447,A -12.523,B 90.000,C 0.000} C_DIS
LIN {X -283.078,Y 62.983,Z 189.176,A -12.544,B 90.000,C 0.000} C_DIS
LIN {X -283.069,Y 63.024,Z 188.562,A -12.552,B 90.000,C 0.000} C_DIS
LIN {X -283.047,Y 63.124,Z 188.291,A -12.572,B 90.000,C 0.000} C_DIS
LIN {X -283.038,Y 63.165,Z 187.568,A -12.580,B 90.000,C 0.000} C_DIS
LIN {X -283.015,Y 63.265,Z 187.279,A -12.601,B 90.000,C 0.000} C_DIS
LIN {X -283.006,Y 63.306,Z 186.557,A -12.609,B 90.000,C 0.000} C_DIS
LIN {X -282.984,Y 63.406,Z 186.286,A -12.629,B 90.000,C 0.000} C_DIS
LIN {X -282.974,Y 63.447,Z 185.671,A -12.638,B 90.000,C 0.000} C_DIS
LIN {X -282.952,Y 63.547,Z 185.400,A -12.658,B 90.000,C 0.000} C_DIS
LIN {X -282.943,Y 63.588,Z 184.678,A -12.666,B 90.000,C 0.000} C_DIS
LIN {X -282.920,Y 63.688,Z 184.389,A -12.686,B 90.000,C 0.000} C_DIS
LIN {X -282.911,Y 63.729,Z 183.666,A -12.695,B 90.000,C 0.000} C_DIS
LIN {X -282.888,Y 63.829,Z 183.395,A -12.715,B 90.000,C 0.000} C_DIS
LIN {X -282.879,Y 63.870,Z 182.781,A -12.723,B 90.000,C 0.000} C_DIS
LIN {X -282.856,Y 63.970,Z 182.510,A -12.744,B 90.000,C 0.000} C_DIS
LIN {X -282.847,Y 64.011,Z 181.787,A -12.752,B 90.000,C 0.000} C_DIS
LIN {X -282.825,Y 64.111,Z 181.498,A -12.772,B 90.000,C 0.000} C_DIS
LIN {X -282.815,Y 64.152,Z 180.775,A -12.780,B 90.000,C 0.000} C_DIS
LIN {X -282.793,Y 64.252,Z 180.505,A -12.801,B 90.000,C 0.000} C_DIS
LIN {X -282.783,Y 64.293,Z 179.890,A -12.809,B 90.000,C 0.000} C_DIS
LIN {X -282.761,Y 64.393,Z 179.619,A -12.829,B 90.000,C 0.000} C_DIS
LIN {X -282.751,Y 64.433,Z 178.897,A -12.837,B 90.000,C 0.000} C_DIS
LIN {X -282.728,Y 64.534,Z 178.608,A -12.858,B 90.000,C 0.000} C_DIS
LIN {X -282.719,Y 64.574,Z 177.885,A -12.866,B 90.000,C 0.000} C_DIS
LIN {X -282.696,Y 64.675,Z 177.614,A -12.886,B 90.000,C 0.000} C_DIS
LIN {X -282.687,Y 64.716,Z 177.000,A -12.895,B 90.000,C 0.000} C_DIS
LIN {X -282.664,Y 64.816,Z 176.729,A -12.915,B 90.000,C 0.000} C_DIS
LIN {X -282.655,Y 64.856,Z 176.006,A -12.923,B 90.000,C 0.000} C_DIS
LIN {X -282.632,Y 64.956,Z 175.735,A -12.943,B 90.000,C 0.000} C_DIS
LIN {X -282.622,Y 64.997,Z 175.121,A -12.952,B 90.000,C 0.000} C_DIS
LIN {X -282.599,Y 65.098,Z 174.850,A -12.972,B 90.000,C 0.000} C_DIS
LIN {X -282.590,Y 65.138,Z 174.127,A -12.980,B 90.000,C 0.000} C_DIS
LIN {X -282.567,Y 65.238,Z 173.838,A -13.001,B 90.000,C 0.000} C_DIS
LIN {X -282.557,Y 65.279,Z 173.115,A -13.009,B 90.000,C 0.000} C_DIS
LIN {X -282.534,Y 65.379,Z 172.826,A -13.029,B 90.000,C 0.000} C_DIS
LIN {X -282.525,Y 65.419,Z 172.104,A -13.037,B 90.000,C 0.000} C_DIS
LIN {X -282.502,Y 65.520,Z 171.833,A -13.058,B 90.000,C 0.000} C_DIS
LIN {X -282.492,Y 65.561,Z 171.219,A -13.066,B 90.000,C 0.000} C_DIS
LIN {X -282.469,Y 65.661,Z 170.948,A -13.086,B 90.000,C 0.000} C_DIS
LIN {X -282.460,Y 65.701,Z 170.225,A -13.094,B 90.000,C 0.000} C_DIS
LIN {X -282.436,Y 65.801,Z 169.954,A -13.115,B 90.000,C 0.000} C_DIS
LIN {X -282.427,Y 65.842,Z 169.340,A -13.123,B 90.000,C 0.000} C_DIS
LIN {X -282.403,Y 65.942,Z 169.069,A -13.143,B 90.000,C 0.000} C_DIS
LIN {X -282.394,Y 65.983,Z 168.346,A -13.151,B 90.000,C 0.000} C_DIS
LIN {X -282.370,Y 66.083,Z 168.057,A -13.172,B 90.000,C 0.000} C_DIS
LIN {X -282.361,Y 66.123,Z 167.334,A -13.180,B 90.000,C 0.000} C_DIS
LIN {X -282.338,Y 66.223,Z 167.063,A -13.200,B 90.000,C 0.000} C_DIS
LIN {X -282.328,Y 66.264,Z 166.449,A -13.209,B 90.000,C 0.000} C_DIS
LIN {X -282.304,Y 66.364,Z 166.178,A -13.229,B 90.000,C 0.000} C_DIS
LIN {X -282.295,Y 66.405,Z 165.456,A -13.237,B 90.000,C 0.000} C_DIS
LIN {X -282.271,Y 66.505,Z 165.166,A -13.258,B 90.000,C 0.000} C_DIS
LIN {X -282.262,Y 66.545,Z 164.444,A -13.266,B 90.000,C 0.000} C_DIS
LIN {X -282.238,Y 66.645,Z 164.173,A -13.286,B 90.000,C 0.000} C_DIS
LIN {X -282.228,Y 66.686,Z 163.559,A -13.294,B 90.000,C 0.000} C_DIS
LIN {X -282.205,Y 66.786,Z 163.288,A -13.315,B 90.000,C 0.000} C_DIS
LIN {X -282.195,Y 66.827,Z 162.565,A -13.323,B 90.000,C 0.000} C_DIS
LIN {X -282.172,Y 66.927,Z 162.276,A -13.343,B 90.000,C 0.000} C_DIS
LIN {X -282.162,Y 66.967,Z 161.553,A -13.351,B 90.000,C 0.000} C_DIS
LIN {X -282.138,Y 67.067,Z 161.282,A -13.372,B 90.000,C 0.000} C_DIS
LIN {X -282.128,Y 67.108,Z 160.668,A -13.380,B 90.000,C 0.000} C_DIS
LIN {X -282.105,Y 67.208,Z 160.397,A -13.400,B 90.000,C 0.000} C_DIS
LIN {X -282.095,Y 67.248,Z 159.674,A -13.408,B 90.000,C 0.000} C_DIS
LIN {X -282.071,Y 67.349,Z 159.385,A -13.429,B 90.000,C 0.000} C_DIS
LIN {X -282.062,Y 67.389,Z 158.663,A -13.437,B 90.000,C 0.000} C_DIS
LIN {X -282.038,Y 67.489,Z 158.392,A -13.457,B 90.000,C 0.000} C_DIS
LIN {X -282.028,Y 67.530,Z 157.777,A -13.466,B 90.000,C 0.000} C_DIS
LIN {X -282.004,Y 67.630,Z 157.506,A -13.486,B 90.000,C 0.000} C_DIS
LIN {X -281.994,Y 67.670,Z 156.784,A -13.494,B 90.000,C 0.000} C_DIS
LIN {X -281.970,Y 67.770,Z 156.513,A -13.514,B 90.000,C 0.000} C_DIS
LIN {X -281.960,Y 67.811,Z 155.899,A -13.523,B 90.000,C 0.000} C_DIS
LIN {X -281.948,Y 67.861,Z 155.772,A -13.533,B 90.000,C 0.000} C_DIS
LIN {X -280.004,Y 67.393,Z 155.772,A -13.533,B 90.000,C 0.000} C_DIS
WAIT SEC 0.1
RET=EKI_SetBool("oxy","torchState",FALSE)
RET = EKI_Send("oxy","torchState")
LIN {X -262.504,Y 63.181,Z 155.772,A -13.533,B 90.000,C 0.000} C_DIS
LIN {X -269.900,Y 7.353,Z 104.656,A -1.561,B 90.000,C 0.000} C_DIS
LIN {X -287.893,Y 7.844,Z 104.656,A -1.561,B 90.000,C 0.000} C_DIS
LIN {X -289.892,Y 7.898,Z 104.656,A -1.561,B 90.000,C 0.000} C_DIS
WAIT SEC 1
RET=EKI_SetBool("oxy","torchState",TRUE)
RET = EKI_Send("oxy","torchState")
LIN {X -289.895,Y 7.807,Z 104.723,A -1.543,B 90.000,C 0.000} C_DIS
LIN {X -289.897,Y 7.735,Z 104.716,A -1.528,B 90.000,C 0.000} C_DIS
LIN {X -289.897,Y 7.726,Z 104.668,A -1.527,B 90.000,C 0.000} C_DIS
LIN {X -289.896,Y 7.775,Z 104.629,A -1.536,B 90.000,C 0.000} C_DIS
LIN {X -289.894,Y 7.839,Z 104.545,A -1.549,B 90.000,C 0.000} C_DIS
LIN {X -289.893,Y 7.886,Z 104.238,A -1.558,B 90.000,C 0.000} C_DIS
LIN {X -289.891,Y 7.937,Z 104.176,A -1.568,B 90.000,C 0.000} C_DIS
LIN {X -289.890,Y 7.988,Z 104.133,A -1.578,B 90.000,C 0.000} C_DIS
LIN {X -289.889,Y 8.031,Z 103.929,A -1.587,B 90.000,C 0.000} C_DIS
LIN {X -289.887,Y 8.082,Z 103.887,A -1.597,B 90.000,C 0.000} C_DIS
LIN {X -289.886,Y 8.133,Z 103.823,A -1.607,B 90.000,C 0.000} C_DIS
LIN {X -289.885,Y 8.175,Z 103.517,A -1.615,B 90.000,C 0.000} C_DIS
LIN {X -289.883,Y 8.226,Z 103.453,A -1.626,B 90.000,C 0.000} C_DIS
LIN {X -289.882,Y 8.277,Z 103.411,A -1.636,B 90.000,C 0.000} C_DIS
LIN {X -289.881,Y 8.320,Z 103.206,A -1.644,B 90.000,C 0.000} C_DIS
LIN {X -289.879,Y 8.371,Z 103.164,A -1.654,B 90.000,C 0.000} C_DIS
LIN {X -289.878,Y 8.422,Z 103.100,A -1.664,B 90.000,C 0.000} C_DIS
LIN {X -289.876,Y 8.464,Z 102.794,A -1.673,B 90.000,C 0.000} C_DIS
LIN {X -289.875,Y 8.515,Z 102.730,A -1.683,B 90.000,C 0.000} C_DIS
LIN {X -289.873,Y 8.566,Z 102.688,A -1.693,B 90.000,C 0.000} C_DIS
LIN {X -289.872,Y 8.609,Z 102.484,A -1.701,B 90.000,C 0.000} C_DIS
LIN {X -289.871,Y 8.660,Z 102.441,A -1.711,B 90.000,C 0.000} C_DIS
LIN {X -289.869,Y 8.711,Z 102.378,A -1.721,B 90.000,C 0.000} C_DIS
LIN {X -289.868,Y 8.753,Z 102.071,A -1.730,B 90.000,C 0.000} C_DIS
LIN {X -289.866,Y 8.804,Z 102.008,A -1.740,B 90.000,C 0.000} C_DIS
LIN {X -289.865,Y 8.855,Z 101.965,A -1.750,B 90.000,C 0.000} C_DIS
LIN {X -289.863,Y 8.898,Z 101.761,A -1.758,B 90.000,C 0.000} C_DIS
LIN {X -289.862,Y 8.949,Z 101.719,A -1.768,B 90.000,C 0.000} C_DIS
LIN {X -289.860,Y 9.000,Z 101.655,A -1.778,B 90.000,C 0.000} C_DIS
LIN {X -289.859,Y 9.042,Z 101.349,A -1.787,B 90.000,C 0.000} C_DIS
LIN {X -289.857,Y 9.093,Z 101.285,A -1.797,B 90.000,C 0.000} C_DIS
LIN {X -289.856,Y 9.144,Z 101.243,A -1.807,B 90.000,C 0.000} C_DIS
LIN {X -289.854,Y 9.187,Z 101.038,A -1.815,B 90.000,C 0.000} C_DIS
LIN {X -289.853,Y 9.238,Z 100.996,A -1.825,B 90.000,C 0.000} C_DIS
LIN {X -289.851,Y 9.289,Z 100.932,A -1.835,B 90.000,C 0.000} C_DIS
LIN {X -289.850,Y 9.331,Z 100.626,A -1.844,B 90.000,C 0.000} C_DIS
LIN {X -289.848,Y 9.382,Z 100.562,A -1.854,B 90.000,C 0.000} C_DIS
LIN {X -289.847,Y 9.433,Z 100.520,A -1.864,B 90.000,C 0.000} C_DIS
LIN {X -289.845,Y 9.476,Z 100.316,A -1.872,B 90.000,C 0.000} C_DIS
LIN {X -289.843,Y 9.527,Z 100.273,A -1.883,B 90.000,C 0.000} C_DIS
LIN {X -289.842,Y 9.578,Z 100.210,A -1.893,B 90.000,C 0.000} C_DIS
LIN {X -289.840,Y 9.620,Z 99.903,A -1.901,B 90.000,C 0.000} C_DIS
LIN {X -289.839,Y 9.671,Z 99.840,A -1.911,B 90.000,C 0.000} C_DIS
LIN {X -289.837,Y 9.722,Z 99.797,A -1.921,B 90.000,C 0.000} C_DIS
LIN {X -289.836,Y 9.764,Z 99.593,A -1.930,B 90.000,C 0.000} C_DIS
LIN {X -289.834,Y 9.815,Z 99.551,A -1.940,B 90.000,C 0.000} C_DIS
LIN {X -289.832,Y 9.866,Z 99.487,A -1.950,B 90.000,C 0.000} C_DIS
LIN {X -289.831,Y 9.909,Z 99.181,A -1.958,B 90.000,C 0.000} C_DIS
LIN {X -289.829,Y 9.960,Z 99.117,A -1.968,B 90.000,C 0.000} C_DIS
LIN {X -289.827,Y 10.011,Z 99.075,A -1.978,B 90.000,C 0.000} C_DIS
LIN {X -289.826,Y 10.053,Z 98.871,A -1.987,B 90.000,C 0.000} C_DIS
LIN {X -289.824,Y 10.104,Z 98.828,A -1.997,B 90.000,C 0.000} C_DIS
LIN {X -289.822,Y 10.155,Z 98.764,A -2.007,B 90.000,C 0.000} C_DIS
LIN {X -289.821,Y 10.198,Z 98.458,A -2.015,B 90.000,C 0.000} C_DIS
LIN {X -289.819,Y 10.249,Z 98.395,A -2.025,B 90.000,C 0.000} C_DIS
LIN {X -289.817,Y 10.300,Z 98.352,A -2.035,B 90.000,C 0.000} C_DIS
LIN {X -289.816,Y 10.342,Z 98.148,A -2.044,B 90.000,C 0.000} C_DIS
LIN {X -289.814,Y 10.393,Z 98.105,A -2.054,B 90.000,C 0.000} C_DIS
LIN {X -289.812,Y 10.444,Z 98.042,A -2.064,B 90.000,C 0.000} C_DIS
LIN {X -289.810,Y 10.487,Z 97.736,A -2.072,B 90.000,C 0.000} C_DIS
LIN {X -289.807,Y 10.589,Z 97.608,A -2.092,B 90.000,C 0.000} C_DIS
LIN {X -289.805,Y 10.631,Z 97.302,A -2.101,B 90.000,C 0.000} C_DIS
LIN {X -289.803,Y 10.682,Z 97.238,A -2.111,B 90.000,C 0.000} C_DIS
LIN {X -289.801,Y 10.733,Z 97.196,A -2.121,B 90.000,C 0.000} C_DIS
LIN {X -289.800,Y 10.775,Z 96.992,A -2.129,B 90.000,C 0.000} C_DIS
LIN {X -289.798,Y 10.826,Z 96.949,A -2.140,B 90.000,C 0.000} C_DIS
LIN {X -289.796,Y 10.877,Z 96.886,A -2.150,B 90.000,C 0.000} C_DIS
LIN {X -289.794,Y 10.920,Z 96.579,A -2.158,B 90.000,C 0.000} C_DIS
LIN {X -289.792,Y 10.971,Z 96.516,A -2.168,B 90.000,C 0.000} C_DIS
LIN {X -289.790,Y 11.022,Z 96.473,A -2.178,B 90.000,C 0.000} C_DIS
LIN {X -289.789,Y 11.064,Z 96.269,A -2.187,B 90.000,C 0.000} C_DIS
LIN {X -289.787,Y 11.115,Z 96.227,A -2.197,B 90.000,C 0.000} C_DIS
LIN {X -289.785,Y 11.166,Z 96.163,A -2.207,B 90.000,C 0.000} C_DIS
LIN {X -289.783,Y 11.209,Z 95.857,A -2.215,B 90.000,C 0.000} C_DIS
LIN {X -289.781,Y 11.260,Z 95.793,A -2.225,B 90.000,C 0.000} C_DIS
LIN {X -289.779,Y 11.311,Z 95.751,A -2.235,B 90.000,C 0.000} C_DIS
LIN {X -289.778,Y 11.353,Z 95.546,A -2.244,B 90.000,C 0.000} C_DIS
LIN {X -289.776,Y 11.404,Z 95.504,A -2.254,B 90.000,C 0.000} C_DIS
LIN {X -289.774,Y 11.455,Z 95.440,A -2.264,B 90.000,C 0.000} C_DIS
LIN {X -289.772,Y 11.498,Z 95.134,A -2.272,B 90.000,C 0.000} C_DIS
LIN {X -289.770,Y 11.549,Z 95.070,A -2.282,B 90.000,C 0.000} C_DIS
LIN {X -289.768,Y 11.600,Z 95.028,A -2.292,B 90.000,C 0.000} C_DIS
LIN {X -289.766,Y 11.642,Z 94.824,A -2.301,B 90.000,C 0.000} C_DIS
LIN {X -289.764,Y 11.693,Z 94.781,A -2.311,B 90.000,C 0.000} C_DIS
LIN {X -289.762,Y 11.744,Z 94.718,A -2.321,B 90.000,C 0.000} C_DIS
LIN {X -289.760,Y 11.786,Z 94.411,A -2.329,B 90.000,C 0.000} C_DIS
LIN {X -289.758,Y 11.837,Z 94.348,A -2.339,B 90.000,C 0.000} C_DIS
LIN {X -289.756,Y 11.888,Z 94.305,A -2.349,B 90.000,C 0.000} C_DIS
LIN {X -289.754,Y 11.931,Z 94.101,A -2.358,B 90.000,C 0.000} C_DIS
LIN {X -289.752,Y 11.982,Z 94.059,A -2.368,B 90.000,C 0.000} C_DIS
LIN {X -289.750,Y 12.033,Z 93.995,A -2.378,B 90.000,C 0.000} C_DIS
LIN {X -289.748,Y 12.075,Z 93.689,A -2.386,B 90.000,C 0.000} C_DIS
LIN {X -289.746,Y 12.126,Z 93.625,A -2.396,B 90.000,C 0.000} C_DIS
LIN {X -289.744,Y 12.177,Z 93.583,A -2.407,B 90.000,C 0.000} C_DIS
LIN {X -289.742,Y 12.220,Z 93.378,A -2.415,B 90.000,C 0.000} C_DIS
LIN {X -289.740,Y 12.271,Z 93.336,A -2.425,B 90.000,C 0.000} C_DIS
LIN {X -289.738,Y 12.322,Z 93.272,A -2.435,B 90.000,C 0.000} C_DIS
LIN {X -289.736,Y 12.364,Z 92.966,A -2.444,B 90.000,C 0.000} C_DIS
LIN {X -289.734,Y 12.415,Z 92.902,A -2.454,B 90.000,C 0.000} C_DIS
LIN {X -289.732,Y 12.466,Z 92.860,A -2.464,B 90.000,C 0.000} C_DIS
LIN {X -289.730,Y 12.508,Z 92.656,A -2.472,B 90.000,C 0.000} C_DIS
LIN {X -289.728,Y 12.559,Z 92.613,A -2.482,B 90.000,C 0.000} C_DIS
LIN {X -289.726,Y 12.610,Z 92.550,A -2.492,B 90.000,C 0.000} C_DIS
LIN {X -289.724,Y 12.653,Z 92.243,A -2.501,B 90.000,C 0.000} C_DIS
LIN {X -289.722,Y 12.704,Z 92.180,A -2.511,B 90.000,C 0.000} C_DIS
LIN {X -289.719,Y 12.755,Z 92.137,A -2.521,B 90.000,C 0.000} C_DIS
LIN {X -289.718,Y 12.797,Z 91.933,A -2.529,B 90.000,C 0.000} C_DIS
LIN {X -289.715,Y 12.848,Z 91.891,A -2.539,B 90.000,C 0.000} C_DIS
LIN {X -289.713,Y 12.899,Z 91.827,A -2.549,B 90.000,C 0.000} C_DIS
